//		'DECLARE @ID_INSERTED TABLE (Id INT) INSERT INTO ProductionMachineParameters (IdLineStation, MachineNumber, IdComposedPart, ParamsData, CRC_Sum) OUTPUT INSERTED.ID INTO @ID_INSERTED VALUES ({IdLineStation}, {MachineNumber}, {IdComposedPart}, ( CONVERT ( VARBINARY({iStructDataSize}), {astStructRawData}) ), {iCRC16sum}) SELECT Id FROM @ID_INSERTED';
//		'DECLARE @ID_INSERTED TABLE (Id INT) INSERT INTO ProductionMachineParameters (IdLineStation, MachineNumber, IdComposedPart, ParamsData, CRC_Sum) OUTPUT INSERTED.ID INTO @ID_INSERTED VALUES ({IdLineStation}, {MachineNumber}, (SELECT IdOutComposedPart FROM ProductionLineStation WHERE Id ={IdLineStation}), {astStructRawData}, {iCRC16sum}) SELECT Id FROM @ID_INSERTED';
//		'DECLARE @ID_INSERTED TABLE (Id INT) INSERT INTO ProductionMachineParameters (IdLineStation, MachineNumber, IdComposedPart, ParamsData, CRC_Sum) OUTPUT INSERTED.ID INTO @ID_INSERTED VALUES ({IdLineStation}, {MachineNumber}, (SELECT IdOutComposedPart FROM ProductionLineStation WHERE Id ={IdLineStation}), CAST({astStructRawData} AS VARBINARY({iStructDataSize})), {iCRC16sum}) SELECT Id FROM @ID_INSERTED';
//		'DECLARE @ID_INSERTED TABLE (Id INT) INSERT INTO ProductionMachineParameters (IdLineStation, MachineNumber, IdComposedPart, ParamsData, CRC_Sum) OUTPUT INSERTED.ID INTO @ID_INSERTED VALUES ({IdLineStation}, {MachineNumber}, {IdComposedPart}, {astStructRawData}, {iCRC16sum}) SELECT Id FROM @ID_INSERTED';
//		'DECLARE @ID_INSERTED TABLE (Id INT) INSERT INTO ProductionMachineParameters (IdLineStation, MachineNumber, IdComposedPart, ParamsData, CRC_Sum) OUTPUT INSERTED.ID INTO @ID_INSERTED VALUES ({IdLineStation}, {MachineNumber}, {IdComposedPart}, CAST({astStructRawData} AS VARBINARY({iStructDataSize})), {iCRC16sum}) SELECT Id FROM @ID_INSERTED';
//		'UPDATE [dbo].[ProductionMachineParameters] SET Active = 0 WHERE IdLineStation = {IdLineStation} AND IdComposedPart = {IdComposedPart} DECLARE @ID_INSERTED TABLE (Id INT) INSERT INTO [dbo].[ProductionMachineParameters] (IdLineStation, MachineNumber, IdComposedPart,ParamsData,CRC_Sum,ParamsSizeInBytes) OUTPUT INSERTED.ID INTO @ID_INSERTED VALUES ({IdLineStation}, {MachineNumber}, {IdComposedPart}), CAST( {astStructRawData} AS VARBINARY(';
	
		stSqlComandData.pReturnedData := ADR(diMachineParamsInsertId);
		stSqlComandData.uiReturnedDataSize := SIZEOF(diMachineParamsInsertId);
		stSqlComandData.bSQL_OK := stSqlComandData.bSQL_Done := FALSE;
		// Próba dodania komendy do kolejki
		IF I_SqlCore <> 0 AND_THEN I_SqlCore.mAddCmdToQueue(ADR(stSqlComandData)) THEN
			bCmdSended := bReturnDataBusy := bReturnDataReserved_InsMachParams := TRUE;		// Zajęcie struktury danych
			diMachineParamsInsertId := 0;
		ELSE
			bResultOk := FALSE;
			nErrorID:=nPIM_ErrorCodes.ParamsSaveToDB_Error;
			m_SqlInsMachineParamsData := bCmdAddError := TRUE;
		END_IF
	ELSIF stSqlComandData.bSQL_Done THEN
		IF stSqlComandData.bSQL_OK THEN
			diParamsId := diMachineParamsInsertId;
		ELSE
			nErrorID:=nPIM_ErrorCodes.ParamsSaveToDB_Error;
		END_IF
		bInsMachineParamsData := TRUE;	// Odśwież parametrów w strukturze PIM, skasowanie zmiennej bCmdSended
		bResultOK := stSqlComandData.bSQL_OK;
		m_SqlInsMachineParamsData := bUpdateData := TRUE;
	END_IF
END_IF
bProcessing := bCmdSended AND NOT stSqlComandData.bSQL_Done;
END_METHOD

// Zapis do DB statusu ostatniej operacji - gdy rozkaz zostanie wykonany zwraca TRUE
METHOD m_SqlSelInsStatus : BOOL
VAR_INPUT
	bStatus:BOOL:= FALSE;		// Status operacji do zapisania
	sErrCode:STRING(10);		// kod błędu - tylko jeśli status  FALSE
	bSustein:BOOL:= FALSE;		// Jeśli TRUE po wywołaniu przez FbMaszyny wykonwyanie rozkazu przerzucone na fbStation (wysyłanie rozkazu w tle)- ustawiana odpowiednia flaga 
END_VAR
VAR_OUTPUT
	bProcessing:BOOL;			// Przetwarzanie rozkazu trwa (rozkaz dodany do kolejki)
	bResultOK:BOOL;				// Wynik wykonania rozkazu (do sprawdzenia gdy metoda zwróci TRUE)
	liStatusId:LINT;			// Id statusu części w DB
END_VAR

VAR
	byStatus: BYTE;
	byIsHidden: BYTE;
END_VAR
// Rezerwacja struktury danych dla zapytania
IF NOT bReturnDataBusy OR bReturnDataReserved_InsOperStat AND stRetDataLineStation.IdStacji <> 0 THEN
	IF NOT bCmdSended THEN	// Przygotowanie danych do zapytania
		stSqlComandData.nCmdState:= nSQL_CmdExecState.New;
		stSqlComandData.nCmdType:=nSQL_CmdTypes.SelInsStatusOfOperation;
		stSqlComandData.byExecutingNodeNb:=0;
		stSqlComandData.bWaitForDataReturn:=TRUE;
	
		stSqlComandData.stStatusSaveParams.didLineStation := stRetDataLineStation.IdStacji;
		stSqlComandData.stStatusSaveParams.byStatus := BOOL_TO_BYTE(bStatus);
		IF bStatus THEN
			stSqlComandData.stStatusSaveParams.byIsHidden := BOOL_TO_BYTE(bIsHidden);
		ELSE
			stSqlComandData.stStatusSaveParams.byIsHidden := 0;
		END_IF
		stSqlComandData.stStatusSaveParams.byIsTestMode := BOOL_TO_BYTE(stPimInOut.bTestMode);
		stSqlComandData.stStatusSaveParams.iMachineNb := iMachineNumber;
		stSqlComandData.stStatusSaveParams.lrQuantity := 1.0;
		byStatus := BOOL_TO_BYTE(bStatus);
		byIsHidden := BOOL_TO_BYTE(bIsHidden);
(*		IF bStatus THEN
			sFormat := 'DECLARE @ID_TABLE TABLE (Id bigint) insert into [dbo].[ProductionMachinePartsStatuses] (IdLineStation, Status, MachineNumber, IsHidden) output inserted.id into @ID_TABLE values (%d, %d, %d, %d) SELECT Top(1) Id FROM @ID_TABLE';
				fbFormatStr2(pFormatString := ADR(sFormat),
				arg1:= F_DINT(stRetDataLineStation.IdStacji),
				arg2:= F_BYTE(byStatus),
				arg3:= F_INT(iMachineNumber),
				arg4:= F_BYTE(byIsHidden),
				pDstString := ADR(stSqlComandData.sCmdExpression), nDstSize := SIZEOF(stSqlComandData.sCmdExpression));
		ELSE
			sFormat := 'DECLARE @ID_TABLE TABLE (Id bigint) insert into [dbo].[ProductionMachinePartsStatuses] (IdLineStation, Status, MachineNumber, IsHidden) output inserted.id into @ID_TABLE values (%d, %d, %d, %d) DECLARE @statusId bigint = (SELECT Top(1) Id FROM @ID_TABLE) INSERT INTO [dbo].[ProductionMachinePartsStatusDefectRelation] (IdPartStatus, IdMachineError) values (@statusId, (SELECT Id FROM [dbo].[ProductionMachineError] WHERE Active = 1 AND Code = $'%s$')) SELECT @statusId';
				fbFormatStr2(pFormatString := ADR(sFormat),
				arg1:= F_DINT(stRetDataLineStation.IdStacji),
				arg2:= F_BYTE(byStatus),
				arg3:= F_INT(iMachineNumber),
				arg4:= F_BYTE(byIsHidden),
				arg5:= F_STRINGEx(sErrCode),
				pDstString := ADR(stSqlComandData.sCmdExpression), nDstSize := SIZEOF(stSqlComandData.sCmdExpression));
		END_IF
*)		
		bLastStatus := bStatus;
		sLastErrCode:= sErrCode;
		stSqlComandData.pReturnedData := ADR(liLPartStatusId);
		stSqlComandData.uiReturnedDataSize := SIZEOF(liLPartStatusId);
		bStatusSavedOK := stSqlComandData.bSQL_OK := stSqlComandData.bSQL_Done := FALSE;
		// Próba dodania komendy do kolejki
		IF I_SqlCore <> 0 AND_THEN I_SqlCore.mAddCmdToQueue(ADR(stSqlComandData)) THEN
			bCmdSended := bReturnDataBusy := bReturnDataReserved_InsOperStat := TRUE;		// Zajęcie struktury danych
			liLPartStatusId := 0;
			bInsertStatus S= bSustein;
		ELSE
			bResultOk := FALSE;
			m_SqlSelInsStatus := bCmdAddError := TRUE;
		END_IF
	ELSIF stSqlComandData.bSQL_Done THEN
		IF stSqlComandData.bSQL_OK THEN
			liStatusId := liLPartStatusId;	// Uaktualnij zmienną wyjściową
		END_IF
		bInsertStatus := TRUE;	// Odśwież parametrów w strukturze PIM, skasowanie zmiennej bCmdSended
		bResultOK := stSqlComandData.bSQL_OK;
		m_SqlSelInsStatus := bUpdateData := TRUE;
	END_IF
END_IF
bProcessing := bCmdSended AND NOT stSqlComandData.bSQL_Done;
END_METHOD

// Pobranie z DB statusu ostatniej operacji dla danego DM z poprzedniego stanowiska - gdy rozkaz zostanie wykonany zwraca TRUE
METHOD m_SqlSelLastOperationStatus : BOOL
VAR_INPUT
	sCodeDM:STRING(255);		// Identyfikator części (kod DataMatrix)
END_VAR
VAR_OUTPUT
	bProcessing:BOOL;			// Przetwarzanie rozkazu trwa (rozkaz dodany do kolejki)
	bResultOK:BOOL;				// Wynik wykonania rozkazu (do sprawdzenia gdy metoda zwróci TRUE)
	bPrevOperStat:BOOL;			// Status ostatniej operacji na poprzednim stanowisku
END_VAR
// Rezerwacja struktury danych dla zapytania
IF NOT bReturnDataBusy OR bReturnDataReserved_SelLastOperStat THEN
	IF NOT bCmdSended THEN
		// Przygotowanie danych do zapytania
		stSqlComandData.nCmdState:= nSQL_CmdExecState.New;
		stSqlComandData.nCmdType:=nSQL_CmdTypes.SelLastOperationStatus;
		stSqlComandData.byExecutingNodeNb:=0;
		stSqlComandData.bWaitForDataReturn:=TRUE;

		sFormat := 'SELECT TOP(1) PMPS.Status FROM [dbo].[ProductionMachinePartsStatuses] PMPS INNER JOIN [dbo].[ProductionLineStation] PLS ON PLS.Id = PMPS.IdLineStation WHERE PLS.Active = 1 AND PMPS.NumberId = $'%s$' AND PLS.Name = $'%s$' AND PMPS.IsHidden = 0 ORDER BY PMPS.Date desc';
		fbFormatStr2(pFormatString := ADR(sFormat),
			arg1:= F_STRINGEx(sCodeDM),
			arg2:= F_STRINGEx(sPrevStationName),
			pDstString := ADR(stSqlComandData.sCmdExpression), nDstSize := SIZEOF(stSqlComandData.sCmdExpression));
			
		sLastDMCode := sCodeDM;
		stSqlComandData.pReturnedData := ADR(bPreviousOperationStatus);
		stSqlComandData.uiReturnedDataSize := SIZEOF(bPreviousOperationStatus);
		stSqlComandData.bSQL_OK := stSqlComandData.bSQL_Done := FALSE;
		// Próba dodania komendy do kolejki
		IF I_SqlCore <> 0 AND_THEN I_SqlCore.mAddCmdToQueue(ADR(stSqlComandData)) THEN
			bCmdSended := 	bReturnDataBusy := bReturnDataReserved_SelLastOperStat := TRUE;		// Zajęcie struktury danych
			bPreviousOperationStatus := FALSE;
		ELSE
			bResultOk := FALSE;
			m_SqlSelLastOperationStatus := bCmdAddError := TRUE;
		END_IF
	ELSIF stSqlComandData.bSQL_Done THEN		// Komenda została wykonana, sprawdzenie rezultatu
		IF stSqlComandData.bSQL_OK THEN
			bPrevOperStat := bPreviousOperationStatus;	// Uaktualnij zmienną wyjściową
		END_IF
		bSelPreviousStatus := TRUE;	// Odśwież parametrów w strukturze PIM, skasowanie zmiennej bCmdSended
		bResultOK := stSqlComandData.bSQL_OK;
		m_SqlSelLastOperationStatus := bUpdateData := TRUE;
	END_IF
END_IF
bProcessing := bCmdSended AND NOT stSqlComandData.bSQL_Done;
END_METHOD

// Pobranie z DB ID stanowiska - gdy rozkaz zostanie wykonany zwraca TRUE
METHOD PRIVATE m_SqlSelLineStationId : BOOL
VAR_INPUT
END_VAR
VAR_OUTPUT
	bProcessing:BOOL;			// Przetwarzanie rozkazu trwa (rozkaz dodany do kolejki)
	bResultOK:BOOL;				// Wynik wykonania rozkazu (do sprawdzenia gdy metoda zwróci TRUE)
	diStationId:DINT;			// Identyfikator stanowiska
	liIdCompossedPart:LINT;		// Identyfikator części wyjściowej
	bAutoSaveErrors:BOOL;		// Auto zapis błędów
	bAutoControlMachineParams:BOOL;		// Kontrola parametrów maszyny
	wCrcSumInDB:WORD;			// Suma CRC aktualnych parametrów maszyny dla złożenia wyjściowego
END_VAR
// Rezerwacja struktury danych dla zapytania
IF NOT bReturnDataBusy OR bReturnDataReserved_StationId THEN
	IF NOT bCmdSended THEN
		// Przygotowanie danych do zapytania
		stSqlComandData.nCmdState:= nSQL_CmdExecState.New;
		stSqlComandData.nCmdType:=nSQL_CmdTypes.SelStationId;
		stSqlComandData.byExecutingNodeNb:=0;
		stSqlComandData.bWaitForDataReturn:=TRUE;
		sFormat := 'SELECT PL.Id, PLS.Id, PLS.IsAutoSaveErrors, PLS.IsEol, PLS.IdOutComposedPart, PMP.CRC_Sum, PCP.CodeNumber FROM [dbo].[ProductionLineStation] PLS INNER JOIN [dbo].[ProductionLine] PL on PLS.IdLine=PL.Id LEFT JOIN [dbo].[ProductionMachineParameters] PMP on PLS.Id=PMP.IdLineStation AND PLS.IdOutComposedPart=PMP.IdComposedPart AND PMP.MachineNumber=%d AND PMP.Active=1 LEFT JOIN [dbo].[ProductionComposedPart] PCP on PLS.IdOutComposedPart=PCP.Id AND PCP.Active=1 WHERE PL.Active = 1 AND PL.Name = $'%s$' AND PLS.Name = $'%s$' AND PLS.Active=1';
		fbFormatStr2(pFormatString := ADR(sFormat),
			arg1:= F_INT(iMachineNumber),
			arg2:= F_STRINGEx(sLineName),
			arg3:= F_STRINGEx(sStationName),
			pDstString := ADR(stSqlComandData.sCmdExpression), nDstSize := SIZEOF(stSqlComandData.sCmdExpression));
		stSqlComandData.pReturnedData := ADR(stRetDataLineStation);
		stSqlComandData.uiReturnedDataSize := SIZEOF(stRetDataLineStation);
		stSqlComandData.bSQL_OK := stSqlComandData.bSQL_Done := FALSE;
		// Próba dodania komendy do kolejki
		IF I_SqlCore <> 0 AND_THEN I_SqlCore.mAddCmdToQueue(ADR(stSqlComandData)) THEN
			bSelectStationId := bCmdSended := bReturnDataBusy := bReturnDataReserved_StationId := TRUE;		// Zajęcie struktury danych
			diStationId := 0;
			MEMSET(destAddr := ADR(stRetDataLineStation), n := SIZEOF(stRetDataLineStation), fillByte:= 0);		// Czyszczenie danych 
		ELSE
			bResultOk := FALSE;
			m_SqlSelLineStationId := bCmdAddError := TRUE;
		END_IF
	ELSIF stSqlComandData.bSQL_Done THEN
		IF stSqlComandData.bSQL_OK THEN
			diStationId := stRetDataLineStation.IdStacji;	// Uaktualnij zmienne wyjściowe
			liIdCompossedPart := stRetDataLineStation.IdOutComposedPart;
			bAutoSaveErrors := stRetDataLineStation.AutoSaveErrors;
			bAutoControlMachineParams := FALSE;// stRetDataLineStation.AutoControlMachineParams; 
			wCrcSumInDB:= stRetDataLineStation.CrcSumOfParams;
		END_IF
		bSelectStationId := bUpdateData := TRUE;	// Odświeżenie parametrów w strukturze PIM w cżęści głównej bloku funkcyjnego, skasowanie zmiennej bCmdSended
		bResultOK := stSqlComandData.bSQL_OK;
		m_SqlSelLineStationId := TRUE;
	END_IF
END_IF
bProcessing := bCmdSended AND NOT stSqlComandData.bSQL_Done;
END_METHOD

// Pobranie z DB sumy CRC parametrów pracy maszyny - gdy rozkaz zostanie wykonany zwraca TRUE
METHOD PRIVATE m_SqlSelMachineParamsCRC : BOOL
VAR_INPUT
	liIdCompossedPart:LINT;		// Identyfikator części wyjściowej dla którego powinna zostać pobrana suma 
END_VAR
VAR_OUTPUT
	bProcessing:BOOL;		// Przetwarzanie rozkazu trwa (rozkaz dodany do kolejki)
	bResultOK:BOOL;			// Wynik wykonania rozkazu (do sprawdzenia gdy metoda zwróci TRUE)
	diStationId:DINT;		// Identyfikator stanowiska
	wCrcFromDb:WORD;		// Suma CRC pobrana z DB
END_VAR
// Sprawdzenie danych wejściowych - jeśli błędne przerwij procedure
IF liIdCompossedPart = 0 OR stRetDataLineStation.IdStacji = 0 THEN
	m_SqlSelMachineParamsCRC := TRUE;
	bResultOK := FALSE;
	RETURN;
END_IF

// Rezerwacja struktury danych dla zapytania
IF NOT bReturnDataBusy OR bReturnDataReserved_SelMachParamsCRC THEN
	IF NOT bCmdSended THEN
		// Przygotowanie danych do zapytania
		stSqlComandData.nCmdState:= nSQL_CmdExecState.New;
		stSqlComandData.nCmdType:=nSQL_CmdTypes.SelMachineParamsCRC;
		stSqlComandData.byExecutingNodeNb:=0;
		stSqlComandData.bWaitForDataReturn:=TRUE;
	
		
		sFormat := 'SELECT CRC_Sum, FROM [dbo].[ProductionMachineParameters] WHERE Active = 1 AND IdLineStation = %d AND MachineNumber = %d AND IdComposedPart = %d';
		fbFormatStr2(pFormatString := ADR(sFormat),
			arg1:= F_DINT(stRetDataLineStation.IdStacji),
			arg2:= F_INT(iMachineNumber),
			arg3:= F_LINT(stRetDataLineStation.IdOutComposedPart),
			pDstString := ADR(stSqlComandData.sCmdExpression), nDstSize := SIZEOF(stSqlComandData.sCmdExpression));

(*		stSqlComandData.sCmdExpression := 'SELECT CRC_Sum, FROM [dbo].[ProductionMachineParameters] WHERE Active = 1 AND IdLineStation = {IdLineStation} AND MachineNumber = {MachineNumber} AND IdComposedPart = {IdComposedPart}';
		stSqlComandData.stCmdData.IdLineStation := stRetDataLineStation.IdStacji;
		stSqlComandData.stCmdData.MachineNumber := iMachineNumber;
		IF liIdCompossedPart = 0 THEN			// Jeśli 0 pobiera dla aktualnie produkowanego, można też pobrać dla konkretnego Id
			stSqlComandData.stCmdData.IdComposedPart := stRetDataLineStation.IdOutComposedPart;
		ELSE
			stSqlComandData.stCmdData.IdComposedPart := liIdCompossedPart;
		END_IF	*)
		stSqlComandData.pReturnedData := ADR(wCrcSumInDb);
		stSqlComandData.uiReturnedDataSize := SIZEOF(wCrcSumInDb);
		stSqlComandData.bSQL_OK := stSqlComandData.bSQL_Done := FALSE;
		// Próba dodania komendy do kolejki
		IF I_SqlCore <> 0 AND_THEN I_SqlCore.mAddCmdToQueue(ADR(stSqlComandData)) THEN
			bCmdSended := bReturnDataBusy := bReturnDataReserved_SelMachParamsCRC := TRUE;		// Zajęcie struktury danych
			wCrcSumInDb := 0;
		ELSE
			bResultOk := FALSE;
			m_SqlSelMachineParamsCRC := bCmdAddError := TRUE;
		END_IF
	ELSIF stSqlComandData.bSQL_Done THEN
		IF stSqlComandData.bSQL_OK THEN
			wCrcFromDb := wCrcSumInDb;	// Uaktualnij zmienne wyjściowe
		END_IF
		m_SqlSelMachineParamsCRC := TRUE;	// Odświeżenie parametrów w strukturze PIM w cżęści głównej bloku funkcyjnego, skasowanie zmiennej bCmdSended
		bResultOK := stSqlComandData.bSQL_OK;
		m_SqlSelMachineParamsCRC := bUpdateData := TRUE;
	END_IF
END_IF
bProcessing := bCmdSended AND NOT stSqlComandData.bSQL_Done;
END_METHOD

// Pobranie z DB parametrów pracy maszyny - gdy rozkaz zostanie wykonany zwraca TRUE
METHOD m_SqlSelMachineParamsData : BOOL
VAR_INPUT
	diParamsId:DINT:=0;				// Jeśli 0 - pobiera parametry dla aktualnego złożenia, jeśli <>0 wtedy pobiera zestaw parametrów o danym Id
	pParamsData:POINTER TO BYTE;	// Wskaźnik do struktury parametrów maszyny
	uiParamsDataSize:UINT;			// Rozmiar struktury danych parametrów maszyny
END_VAR
VAR_OUTPUT
	bProcessing:BOOL;				// Przetwarzanie rozkazu trwa (rozkaz dodany do kolejki)
	bResultOK:BOOL;					// Wynik wykonania rozkazu (do sprawdzenia gdy metoda zwróci TRUE)
	bNoMatchingParams:BOOL;			// Błąd - brak pasujących parametrów w DB
	bParametersUpdated:BOOL;		// Parametry maszyny uaktualnione
//	pParamsData: POINTER TO BYTE;
END_VAR
(*
Zapis i odczyt parametrów kontroluje blok klienta PIM, struktura w bloku przechowywana jest jako wskaźnik więc nie jest konieczne powiązanie ze strukturą parametrów maszyny.
Metoda pobiera z DB najnowszy zestaw parametrów lub zestaw o danym Id (jeśli Id nie jest równe 0), sprawdza czy rozmiary oraz suma CRC są zgodne - jeśli są przepisuje pobrane dane do wskaźnika wejściowego.
Jeśli nie co zrobić - może pytanie do użytkownika (przez komendy PIM) "Rozmiar/wartość danych niezgodna - pomiń lub nadpisz" - użytkownik wybierze odpowiendią opcje która zostanie zwrócona do PLC.
Póki co następuje automatyczne przepisanie niekompletnych lub niezgodnych parametrów.
*)

// Sprawdzenie danych wejściowych - jeśli błędne przerwij procedure
IF pParamsData = 0 OR uiParamsDataSize = 0 OR SEL(diParamsId=0, stRetDataLineStation.IdStacji = 0, stRetDataLineStation.IdStacji = 0 OR stRetDataLineStation.IdOutComposedPart = 0) THEN
	m_SqlSelMachineParamsData := TRUE;
	bResultOK := FALSE;
	RETURN;
END_IF

// Rezerwacja struktury danych dla zapytania
IF NOT bReturnDataBusy OR bReturnDataReserved_SelMachParams THEN
	IF NOT bCmdSended THEN	// Przygotowanie danych do zapytania
		stSqlComandData.nCmdState:= nSQL_CmdExecState.New;
		stSqlComandData.nCmdType:=nSQL_CmdTypes.SelMachineParams;
		stSqlComandData.byExecutingNodeNb:=0;
		
	(*	stSqlComandData.bWaitForDataReturn:=TRUE;
		IF diParamsId <> 0 THEN		// Rodzaj zapytania zależy od tego po czym chcemy wyszukiwać zestawy parametrów 
			stSqlComandData.sCmdExpression :=  'SELECT ParamsData, CRC_Sum, ParamsSizeInBytes FROM [dbo].[ProductionMachineParameters] WHERE Id = {IdLineStation}';
			stSqlComandData.stCmdData.IdLineStation := diParamsId;
		ELSE
			stSqlComandData.sCmdExpression :=  'SELECT ParamsData, CRC_Sum, ParamsSizeInBytes FROM [dbo].[ProductionMachineParameters] WHERE Active = 1 AND MachineNumber = {MachineNumber} AND IdLineStation = {IdLineStation} AND IdComposedPart = {IdComposedPart}';
			stSqlComandData.stCmdData.MachineNumber := iMachineNumber;
			stSqlComandData.stCmdData.IdLineStation := stRetDataLineStation.IdStacji;
			stSqlComandData.stCmdData.IdComposedPart := stRetDataLineStation.IdOutComposedPart;
		END_IF	*)
		stSqlComandData.pReturnedData := ADR(stRetDataMachParams);
		stSqlComandData.uiReturnedDataSize := SIZEOF(stRetDataMachParams);
		stSqlComandData.bSQL_OK := stSqlComandData.bSQL_Done := FALSE;
		// Próba dodania komendy do kolejki
		IF I_SqlCore <> 0 AND_THEN  I_SqlCore.mAddCmdToQueue(ADR(stSqlComandData)) THEN
			bCmdSended := bReturnDataBusy := bReturnDataReserved_SelMachParams := TRUE;		// Zajęcie struktury danych
			MEMSET(destAddr := ADR(stRetDataMachParams), n := SIZEOF(stRetDataMachParams), fillByte:= 0);		// Czyszczenie danych 
		ELSE
			bResultOk := FALSE;
			m_SqlSelMachineParamsData := bCmdAddError := TRUE;
		END_IF
	ELSIF stSqlComandData.bSQL_Done THEN	// Przetwarzanie zapytania SQL zakończone 
		IF stSqlComandData.bSQL_OK THEN
			IF stRetDataMachParams.DataSize = UINT_TO_INT(uiParamsDataSize) THEN	// Rozmiar parametrów zgodny
				IF INT_TO_WORD(stRetDataMachParams.CRC16sum) = F_DATA_TO_CRC16_CCITT(pData := ADR(stRetDataMachParams.StructRawData), cbData := INT_TO_UDINT(stRetDataMachParams.DataSize), crc:= 0) THEN
					MEMCPY(srcAddr := ADR(stRetDataMachParams.StructRawData), destAddr := pParamsData, n:= uiParamsDataSize);
					bParametersUpdated := TRUE;
				ELSE		// Niezgodne sumy CRC - raczej niemożliwe
					mNewlnternalEvent(nInputErrorID := nPIM_ErrorCodes.ParamsMismatchPLCandDB, nEventType := nPIM_EventClasses.Alarm, tMessageTime := T#0S);
					MEMCPY(srcAddr := ADR(stRetDataMachParams.StructRawData), destAddr := pParamsData, n:= uiParamsDataSize);
				END_IF
			ELSE
				mNewlnternalEvent(nInputErrorID := nPIM_ErrorCodes.ParamsMismatchPLCandDB, nEventType := nPIM_EventClasses.Alarm, tMessageTime := T#0S);
				MEMSET(destAddr := pParamsData, n := uiParamsDataSize, fillByte:= 0);		// Czyszczenie danych parametrów
				MEMCPY(srcAddr := ADR(stRetDataMachParams.StructRawData), destAddr := pParamsData, n:= MIN(uiParamsDataSize,INT_TO_UINT(stRetDataMachParams.DataSize)));
			END_IF
		ELSE	// Jeśli nie zwrócono żadnego rekordu brak pasujących parametrów - trzeba najpierw przesłać parametry do DB
			mNewlnternalEvent(nInputErrorID := nPIM_ErrorCodes.NoMatchingParamsForComponent, nEventType := nPIM_EventClasses.Alarm, tMessageTime := T#0S);
			bNoMatchingParams := TRUE;	;
		END_IF
		bSelMachineParamsData := TRUE;	// Odświeżenie parametrów w strukturze PIM, skasowanie zmiennej bCmdSended
		bResultOK := stSqlComandData.bSQL_OK;
		m_SqlSelMachineParamsData := bUpdateData := TRUE;
	END_IF
END_IF
pParamsData := ADR(stRetDataMachParams.StructRawData);
bProcessing := bCmdSended AND NOT stSqlComandData.bSQL_Done;
END_METHOD

ACTION ACT_PimCmdsHandling:
// TImer gotowości PIMu (komunikacja itp jest OK)
fbTOF_PimWorking(IN:= FALSE, PT:= T#5M, Q=> bPIM_Working);		// TImer o gotowości systemu PIM

//Obsługa komunikatów z PIMu
IF stPimInOut.sCmdPIM2PLC <> '' AND NOT bCmdReaded THEN
	fbLogger.mAddLine(sTextToSave := CONCAT(STR1:= 'CmdRecived- ', STR2:=stPimInOut.sCmdPIM2PLC));
	sCmdToSendToMachine := sStringToParse := F_ToLCase(stPimInOut.sCmdPIM2PLC);
	WHILE sStringToParse <> '' DO
		sActCmd := fPIM_GetCmdPar(sParseString := sStringToParse);
		IF sActCmd = 'lifebit' THEN
			fbTOF_PimWorking(IN:= TRUE);
		ELSIF sActCmd = 'sendmachineparamstodb' THEN			// Zapisuje w bazie danych parametry pracy dla aktualnego złożenia jako aktywne 
			bMachParamsSendToDB:= TRUE;
		ELSIF sActCmd = 'readmachineparamsfromdb' THEN
			bMachParamsReadFromDB := TRUE;	// Wymuszenie pobrania parametrów z bazy danych
			bMachineParamsOK := FALSE;		// Zatrzymanie pracy na czas pobrania elementów
		ELSIF sActCmd = 'retool' THEN		// Pobiera z bazy danych parametry dla danego złożenia
			sActCmd := fPIM_GetCmdPar(sParseString := sStringToParse);
			liRetoolParamsIdFromPIM:= STRING_TO_LINT(sActCmd);
//			bRetool := TRUE;	// Wymuszenie pobrania parametrów z bazy danych
//			bMachineParamsOK := FALSE;		// Zatrzymanie pracy na czas pobrania elementów
		ELSIF sActCmd = 'newboxout' THEN
			iOutBoxQty:= STRING_TO_INT(fPIM_GetCmdPar(sParseString := sStringToParse));
			iOutBoxTargetQty:= STRING_TO_INT(fPIM_GetCmdPar(sParseString := sStringToParse));
		ELSIF sActCmd = 'nokreported' THEN	// Zgłoszenie po wykonaniu operacji - do ustalenia źródło zgłoszenia
			sActCmd := fPIM_GetCmdPar(sParseString := sStringToParse);				
			IF sActCmd = 'fprevstation' THEN
				nReoprtedNokSource:= nPIM_ReportedNokSource.FromPrevStation;
			ELSIF sActCmd = 'fmach' THEN
				nReoprtedNokSource:= nPIM_ReportedNokSource.FromMach;				
			ELSIF sActCmd = 'fbox' THEN
				nReoprtedNokSource:= nPIM_ReportedNokSource.FromBox;
			ELSE
				nReoprtedNokSource:= nPIM_ReportedNokSource.Error_UnknownSource;			
			END_IF
		ELSIF sActCmd = 'rework' THEN
			IF fPIM_GetCmdPar(sParseString := sStringToParse) = 'true' THEN
				nReworkMenuStatus := nPIM_ReworkSelect.yes;
				iCtr_PIM_ReworkYes := iCtr_PIM_ReworkYes + 1;
				iCtr_PIM_PartsNOK := LIMIT(0,iCtr_PIM_PartsNOK - 1,32767);
			ELSE
				nReworkMenuStatus := nPIM_ReworkSelect.no;
			END_IF
		ELSIF sActCmd = 'logged' THEN
			sUserRole:= fPIM_GetCmdPar(sParseString := sStringToParse);
			sUserLang:= fPIM_GetCmdPar(sParseString := sStringToParse);
		ELSIF sActCmd = '' THEN
			MEMMOVE(srcAddr := ADR(asUnsuportedCmds[1]), destAddr := ADR(asUnsuportedCmds[2]), n := 4*SIZEOF(asUnsuportedCmds[1]));
			asUnsuportedCmds[1] := 'EmptyString';
		ELSE
			MEMMOVE(srcAddr := ADR(asUnsuportedCmds[1]), destAddr := ADR(asUnsuportedCmds[2]), n := 4*SIZEOF(asUnsuportedCmds[1]));
			asUnsuportedCmds[1] := sActCmd;
		END_IF
	END_WHILE
	bCmdReaded := TRUE;
ELSE
	stPimInOut.sCmdPIM2PLC := '';
	ACT_UpdatePimOutput();
	bCmdReaded := FALSE;
	nReoprtedNokSource:= nPIM_ReportedNokSource.none;
	nReworkMenuStatus := nPIM_ReworkSelect.none;
END_IF

//Obsługa komunikatów z PIMu
fbTON_CmdPLC2PIM_Reset(IN:= stPimInOut.sCmdPLC2PIM <> '', PT:= T#100MS);
IF fbTON_CmdPLC2PIM_Reset.Q THEN
	stPimInOut.sCmdPLC2PIM := '';
	bCmdPlc2PimSended := FALSE;
END_IF
bCmdPlc2PimSended R= stPimInOut.sCmdPLC2PIM = '';

(*	Komendy do wysłania:
	- Wyloguj użytkownika?
	- Zgłoś usterkę maszyny
*)
END_ACTION

ACTION ACT_SqlDataReturnCmd:

{warning 'Uzupełnić działanie LifeBita, Timeoutu'}
fbTON_CmdHangedUp(IN:= bReturnDataBusy AND NOT stSqlComandData.bSQL_Done AND I_SqlCore.IsCoreWork(), PT:= T#20S);
IF fbTON_CmdHangedUp.Q THEN
	fbTON_CmdHangedUp(IN:= FALSE);
	stSqlComandData.bSQL_Done := TRUE;
	stSqlComandData.bSQL_Busy := stSqlComandData.bSQL_OK := FALSE;
	fbLogger.mAppendCurrentLine(bBreakLine := TRUE, sAddSep := '', sAppendText:= CONCAT('Sql command Hungedup, service reset- Cmd State ',INT_TO_STRING(stSqlComandData.nCmdState)));
	uiCtr_CmdReset:= uiCtr_CmdReset +1; 
END_IF

stSqlComandData.bSQL_LifeBit := FALSE;

IF bTestAdditionalErrorSave THEN
	bTestAdditionalErrorSave := bTestResult:= FALSE;
	bTestResult:= m_SqlInsAdditionalError(sErrCode := sLastErrCode);
ELSIF bTestComprAirCtrSave THEN
	bTestComprAirCtrSave := bTestResult:= FALSE;
	bTestResult:= m_SqlInsCompressedAirConsumption(rActCompressedAirConsumption := 9.99);
ELSIF bTestEnergyCtrSave THEN
	bTestEnergyCtrSave := bTestResult:= FALSE;
	bTestResult:= m_SqlInsEnergyConsumption(rActEnergyConsumption := 9.99);
ELSIF bTestDefectRealtionSave THEN
	bTestDefectRealtionSave:= bTestResult := FALSE;
	bTestResult:= m_SqlInsDefectRelation(sErrCode := '54');	
END_IF

// Jeśli chcemy serwisowo sprawdzić działanie funkcji ustawić zmienne wejściowe w odpowiedni sposób oraz ustawić zmienną w If np. bSelectStationId
IF bSelectStationId THEN
	IF NOT bUpdateData THEN
		m_SqlSelLineStationId(bProcessing => bPimCmdProcessing);
	END_IF
	IF stSqlComandData.bSQL_Done THEN
		IF stSqlComandData.bSQL_OK THEN		// Pobranie danych OK
		//	stRetDataLineStation.AutoControlMachineParams := FALSE;
			fbLogger.mAddLine(sTextToSave := CONCAT(STR1:= 'RecvStationId- ', STR2:= DINT_TO_STRING(stRetDataLineStation.IdStacji)));
			stStationStatus.stStationSqlData := stRetDataLineStation; 
		ELSE 
			fbLogger.mAddLine(sTextToSave := 'RecvStationId rvc error');
		END_IF
		bPimCmdProcessing := bCmdSended := bSelectStationId := FALSE;
		bReturnDataBusy := bReturnDataReserved_StationId := FALSE;
	//	MEMSET(destAddr := ADR(stDBCmdData), n := SIZEOF(stDBCmdData), fillByte:= 0);		// Czyszczenie danych zapytania
	ELSIF NOT bPimCmdProcessing THEN
		bCmdSended := bSelectStationId := FALSE;
		bReturnDataBusy := bReturnDataReserved_StationId := FALSE;		
	END_IF
END_IF

IF bInsertStatus THEN 
	IF NOT bUpdateData THEN
		m_SqlSelInsStatus(bStatus:=bLastStatus , sErrCode:= sLastErrCode, bSustein := FALSE, bProcessing => bPimCmdProcessing);
	END_IF
	IF stSqlComandData.bSQL_Done THEN	
		IF stSqlComandData.bSQL_OK THEN
			bStatusSavedOK := TRUE;
		
			iCtr_StatusSaveOK := iCtr_StatusSaveOK + 1; 
			mSendCmdToPIM(sCmd := CONCAT(STR1:='StatusId:', STR2:= LINT_TO_STRING(liLPartStatusId)));
			IF bLastStatus THEN
		
				fbLogger.mAddLine(sTextToSave := CONCAT(STR1:= 'Status OK saved, StatusId- ', STR2:= LINT_TO_STRING(liLPartStatusId)));
				iCtr_PIM_PartsOK := iCtr_PIM_PartsOK +1;
			ELSE
				stPimInOut.sStatusNokAndErrorID := CONCAT(STR1:= LINT_TO_STRING(liLPartStatusId), STR2:= CONCAT(STR1:= ':',STR2:= sLastErrCode));
				fbLogger.mAddLine(sTextToSave := CONCAT(STR1:= 'Status NOK saved, StatusId- ', STR2:= LINT_TO_STRING(liLPartStatusId)));
				iCtr_PIM_PartsNOK := iCtr_PIM_PartsNOK +1;
			END_IF
			IF bLockAfterStatusSave THEN
				IF stPimInOut.sErrorCodePLC = '' THEN
					iConvTMP := nPIM_ErrorCodes.UnKnownLock;
					stPimInOut.sErrorCodePLC := INT_TO_STRING(iConvTMP);
				END_IF
				stPimInOut.bAlarmPLC :=  stPimInOut.bNonBlockingAlarm := FALSE;
				bSaveDefectRelation := stPimInOut.bWorkBlock_PLC := TRUE;				
			END_IF
		ELSE
			iCtr_StatusSaveError := iCtr_StatusSaveError + 1; 
			IF stSqlComandData.udiLEventId <> 0 THEN
				mSendCmdToPIM(sCmd := CONCAT(STR1:= 'StatusSaveError:', STR2:= UDINT_TO_STRING(stSqlComandData.udiLEventId)));
			ELSE
				mSendCmdToPIM(sCmd := 'StatusSaveError');
			END_IF
			IF bLastStatus THEN
				fbLogger.mAddLine(sTextToSave := 'Status OK Save error');
				iCtr_PIM_PartOK_SaveError := iCtr_PIM_PartOK_SaveError +1;
			ELSE
				fbLogger.mAddLine(sTextToSave := 'Status NOK Save error');
				iCtr_PIM_PartNOK_SaveError := iCtr_PIM_PartNOK_SaveError +1;
			END_IF
			IF bLockAfterStatusSave THEN
				IF stPimInOut.sErrorCodePLC = '' THEN
					iConvTMP := nPIM_ErrorCodes.UnKnownLock;
					stPimInOut.sErrorCodePLC := INT_TO_STRING(iConvTMP);
				END_IF
				bSaveDefectRelation := stPimInOut.bWorkBlock_PLC := TRUE;
			END_IF
		END_IF
		bPimCmdProcessing := bLockAfterStatusSave := bCmdSended := bInsertStatus := FALSE;		
		bReturnDataBusy := bReturnDataReserved_InsOperStat := FALSE;
	//	MEMSET(destAddr := ADR(stDBCmdData), n := SIZEOF(stDBCmdData), fillByte:= 0);		// Czyszczenie danych zapytania
	ELSIF NOT bPimCmdProcessing THEN
		bCmdSended := bInsertStatus := FALSE;
		bReturnDataBusy := bReturnDataReserved_InsOperStat := FALSE;
		IF bLockAfterStatusSave THEN
			IF stPimInOut.sErrorCodePLC = '' THEN
				iConvTMP := nPIM_ErrorCodes.UnKnownLock;
				stPimInOut.sErrorCodePLC := INT_TO_STRING(iConvTMP);
			END_IF
			stPimInOut.bAlarmPLC :=  stPimInOut.bNonBlockingAlarm := FALSE;
			stPimInOut.bWorkBlock_PLC := TRUE;		
			bLockAfterStatusSave := FALSE;		
		END_IF
	END_IF
ELSIF bLockAfterStatusSave AND stPimInOut.sErrorCodePLC <> '' THEN
//	{warning 'Wstawić sygnał zwrotny zapisu błędu do PIMu- zapis poprawny gdy nie są pobrane parametry z SQLa'}
	bLockAfterStatusSave := FALSE;
	stPimInOut.bAlarmPLC :=  stPimInOut.bNonBlockingAlarm := FALSE;
	stPimInOut.bWorkBlock_PLC := TRUE;	
END_IF


IF bSelPreviousStatus THEN 
	IF NOT bUpdateData THEN
		m_SqlSelLastOperationStatus(sCodeDM:= sLastDMCode, bProcessing => bPimCmdProcessing);
	END_IF
	IF stSqlComandData.bSQL_Done THEN
		IF  stSqlComandData.bSQL_OK THEN
			bPreviousOperationStatus := bPreviousOperationStatus;		
		END_IF
		bPimCmdProcessing := bCmdSended := bSelPreviousStatus := FALSE;
		bReturnDataBusy := bReturnDataReserved_SelLastOperStat := FALSE;
	ELSIF NOT bPimCmdProcessing THEN
		bCmdSended := bSelPreviousStatus := FALSE;
		bReturnDataBusy := bReturnDataReserved_SelLastOperStat := FALSE;		
	END_IF	
END_IF

IF bSelMachineParamsData THEN
	IF NOT bUpdateData THEN
		m_SqlSelMachineParamsData(diParamsId := 0, pParamsData:= 0, uiParamsDataSize := 0, bProcessing => bPimCmdProcessing);
	END_IF
	IF stSqlComandData.bSQL_Done THEN
		bPimCmdProcessing := bCmdSended := bSelMachineParamsData := FALSE;
		bReturnDataBusy := bReturnDataReserved_SelMachParams := FALSE;
	ELSIF NOT bPimCmdProcessing THEN
		bCmdSended := bSelMachineParamsData := FALSE;
		bReturnDataBusy := bReturnDataReserved_SelMachParams := FALSE;		
	END_IF
END_IF

IF bSelMachineParamsCRC THEN
	IF NOT bUpdateData THEN
		m_SqlSelMachineParamsCRC(liIdCompossedPart := 0, bProcessing => bPimCmdProcessing);
	END_IF
	IF stSqlComandData.bSQL_Done THEN
		IF stSqlComandData.bSQL_OK THEN
			diMachineParamsInsertId := diMachineParamsInsertId;
		END_IF
		bPimCmdProcessing := bCmdSended := bSelMachineParamsCRC := FALSE;
		bReturnDataBusy := bReturnDataReserved_SelMachParamsCRC := FALSE;
	ELSIF NOT bPimCmdProcessing THEN 
		bCmdSended := bSelMachineParamsCRC := FALSE;
		bReturnDataBusy := bReturnDataReserved_SelMachParamsCRC := FALSE;		
	END_IF
END_IF

IF bInsMachineParamsData THEN
	IF NOT bUpdateData THEN
		m_SqlInsMachineParamsData(pParamsData := 0, uiParamsDataSize := 0, wCrcSumOfParameters := 0, bProcessing => bPimCmdProcessing);
	END_IF
	IF stSqlComandData.bSQL_Done THEN
		IF stSqlComandData.bSQL_OK THEN
			diMachineParamsInsertId := diMachineParamsInsertId;
		END_IF
		bPimCmdProcessing := bCmdSended := bInsMachineParamsData := FALSE;
		bReturnDataBusy := bReturnDataReserved_InsMachParams := FALSE;
	ELSIF NOT bPimCmdProcessing THEN 
		bCmdSended := bInsMachineParamsData := FALSE;
		bReturnDataBusy := bReturnDataReserved_InsMachParams := FALSE;		
	END_IF
END_IF


ACT_UpdatePimOutput();
bUpdateData := FALSE;
END_ACTION

ACTION ACT_UpdatePimOutput:
(*
IF stPimInternal.sCmdPLC2PIM <> '' THEN
	stPimInOut.sCmdPLC2PIM := stPimInternal.sCmdPLC2PIM;	
	bCmdPlc2PimSended:= TRUE;
ELSIF sCmdPlc2PimBufer <> '' THEN
	stPimInternal.sCmdPLC2PIM := sCmdPlc2PimBufer; 
	bCmdPlc2PimSended:= TRUE;
ELSIF stPimInternal.sCmdPLC2PIM = '' THEN
	 stPimInOut.sCmdPLC2PIM := '';
END_IF
*)
END_ACTION

METHOD FB_init : BOOL
VAR_INPUT
	bInitRetains : BOOL; // if TRUE, the retain variables are initialized (warm start / cold start)
	bInCopyCode : BOOL;  // if TRUE, the instance afterwards gets moved into the copy code (online change)
	I_Mach: I_StationMachine;				// Interfejs do obsługi maszyn - pobranie danych z maszyny (głównie parametry pracy)
	I_Sql:	I_SQL_Core;		
END_VAR
I_Machine := I_Mach;
I_SqlCore := I_Sql;
END_METHOD

// Metoda zwraca strukturę do zapytania SQL uzupełnioną o dane z bloczka stanowiska
METHOD mGetStationData : stPIM_StationStatus
VAR_OUTPUT
	sCMD				: STRING;		// Zdarzenie jednostkowe/ rozkaz z PIMu np uaktualniono dane itp.
	bUserLogged			: BOOL;			// Użytkownik zalogowany
	bPIM_Active			: BOOL;			// Info o aktywności systemu PIM
	bTestMode			: BOOL;			// Aktywny tryb testowy
	bWorkPermittion		: BOOL;			// Informacja o zezwoleniu na pracę sumarycznie
	bWorkBlockPIM		: BOOL;			// Informacja o zezwoleniu na pracę z PIM
	bWorkBlockPLC		: BOOL;			// Informacja o zezwoleniu na pracę z PLC
	bConfirmation		: BOOL;			// Informacja o potwierdzeniu błędu
	bExternalMessage	: BOOL;			// Informacja o aktywnym komunikacie zewnętrznym
	nExtErrorClass		: nPIM_EventClasses;			// Informacja o aktywnym błędzie zewnętrznym
	bEventWaitInQueue	: BOOL;			// Info, że zdarzenie zewnętrzne czeka w kolejce
	nMachState			: nPIM_MachineStates;	// Aktualny status maszyny
	bOperInProgress		: BOOL;			// TRUE gdy operacja trwa
	bOperEnded			: BOOL;			// Impuls gdy operacja zakończona
	bOperStatus			: BOOL;			// Status ostatniej operacji
	nReworkSelected 	: nPIM_ReworkSelect;	// Operator wybrał Opcje reworku na tak lub nie
	nReoprtedNok 		: nPIM_ReportedNokSource;	// Operator zgłosił NOKa
END_VAR

mGetStationData:= stStationStatus;

sCMD := sCmdToSendToMachine;
sCmdToSendToMachine := '';
bUserLogged := fbTON_UserLogedDeleyed.Q;
bPIM_Active := stPimInOut.bPIMActive;
bWorkPermittion	:= bWorkPermitt;	
bWorkBlockPIM := stPimInOut.bWorkBlock_PIM;
bWorkBlockPLC := stPimInOut.bWorkBlock_PLC;
bConfirmation := stPimInOut.bConfirmEvent;
bTestMode := stPimInOut.bTestMode;
nExtErrorClass := nActExtErrorClass;
nMachState := nMachineState;
bEventWaitInQueue := iNextEventCodeEnum <> 0 AND bNextEventSource;

bOperInProgress := nMachineState = nPIM_MachineStates._4_OperationInProgress ;
bOperEnded := bOperationEnded OR nMachineState = nPIM_MachineStates._5_OperationEndedOK ;
bOperStatus := bLastStatus;
nReworkSelected:= nReworkMenuStatus;
nReoprtedNok := nReoprtedNokSource;
END_METHOD

METHOD PUBLIC mNewEvent : BOOL
VAR_INPUT
	iEventId:	INT;				// Kod błędu w postaci inta (do przekonwertowania)
	nEventType: nPIM_EventClasses;	// ROdzaj nowego zdarzenia
	tMessageTime: TIME:= T#3S;		// Czas na wyświetlenie wiadomości- ma znaczenie tylko dla wiadomości (po tym czasie lub po starcie nowej operacji wiadomość znika)
END_VAR
VAR
	sType: STRING;
END_VAR
// Zgłaszanie błędu zewnętrznego
IF nActIntErrorClass = nPIM_EventClasses.NoError THEN	// Jeśli aktualnienie ma aktywnego błędu dodaj jako podstawowy
	mNewEventCommon(iErrorEnum:= iEventId, nAlarmType := nEventType, tMessageTime := tMessageTime);
	nActExtErrorClass := nEventType;
ELSE	// Jeśli jest aktywny błąd wewnętrzny sprawdź co zrobić
	IF nEventType > nActIntErrorClass THEN	// Błąd zewnętrzny ważniejszy niż aktualny to
		IF nActIntErrorClass > nPIM_EventClasses.Message THEN 	// Jeśli aktywny wewnętrzny błąd ma priorytet wyższy niż wiadomość zamień błąd, a aktywny przenieś co pamięci 
			iNextEventCodeEnum := STRING_TO_INT(stPimInOut.sErrorCodePLC);
			nNextEeventType := nActIntErrorClass;
			bNextEventSource := FALSE;
			nActIntErrorClass := nPIM_EventClasses.NoError;
		ELSE	// Jeśli aktywna jest wiadomość tylko ją nadpisz
			nActIntErrorClass := nPIM_EventClasses.NoError;
			mNewEventCommon(iErrorEnum:= iEventId, nAlarmType := nEventType, tMessageTime := tMessageTime);
			nActExtErrorClass := nEventType;
		END_IF
	ELSE	// Błąd zewnętrzny ma niższy priorytet - dodanie nowego błędu do kolejki
		iNextEventCodeEnum := iEventId;
		nNextEeventType := nEventType;
		tNextEeventMessageTime := tMessageTime;
		bNextEventSource := TRUE;
	END_IF
END_IF

iCtr_NewEventCalls := iCtr_NewEventCalls+1;
IF nEventType = nPIM_EventClasses.Error THEN
	iCtr_NewEventCalls_ER := iCtr_NewEventCalls_ER +1;
ELSIF nEventType = nPIM_EventClasses.Alarm THEN
	iCtr_NewEventCalls_AL := iCtr_NewEventCalls_AL +1;
ELSE
	iCtr_NewEventCalls_Other := iCtr_NewEventCalls_Other +1;	
END_IF

// Logowanie danych
sType:= TO_STRING(nEventType);
fbFormatStr(sFormat := 'Nowy event zewnetrzny typ- %s, Id- %d',
	arg1 := F_STRINGEx(sType), 
	arg2 := F_INT(iEventId));  
fbLogger.mAddLine(sTextToSave := fbFormatStr.sOut );
mNewEvent := TRUE;

(*
IF NOT bInternalEventActive THEN	// Brak aktywnego alarmu lub aktywny alarm zewnętrzny (wtedy zamienia alarm)- dodaj alarm jako podstawowy
	mNewEventCommon(iErrorEnum:= iEventId, nAlarmType := nEventType, tMessageTime := tMessageTime);
	bExternalEventActive := nEventType = nPIM_EventClasses.Error OR nEventType = nPIM_EventClasses.Alarm;
	bExternalMessageActive := NOT bExternalEventActive;
	bInternalMessageActive := FALSE;		// Kasowanie wiadomości wewnętrznej (alarm ma wyższy priorytet
ELSE	// Alarm wewnętrzny jest już wyświetlany, dodaj alarm do kolejki
	
END_IF
*)
END_METHOD

// Kod wspólny dla zgłaszania błędów zewnętrznych i wewnętrznych
METHOD INTERNAL mNewEventCommon : BOOL
VAR_INPUT
	iErrorEnum:	INT;				// Kod błędu w postaci inta (do przekonwertowania)
	nAlarmType: nPIM_EventClasses;	// ROdzaj nowego zdarzenia
	tMessageTime: TIME:= T#3S;		// Czas na wyświetlenie wiadomości- ma znaczenie tylko dla wiadomości (po tym czasie lub po starcie nowej operacji wiadomość znika)
END_VAR
// Akcja z obsługą błędu - zmienne In_Out nie powinny być używane w metodach
// Określenie kodu alarmu
IF iErrorEnum <> 0 THEN		// Kod błędu podany przez Enum
	stPimInOut.sErrorCodePLC := INT_TO_STRING(iErrorEnum);
ELSE	// Brak kodu błędu -
	iConvTMP := nPIM_ErrorCodes.UnKnownLock;
	stPimInOut.sErrorCodePLC := INT_TO_STRING(iConvTMP);
END_IF		
bSaveDefectRelation R= NOT stPimInOut.bWorkBlock_PLC;

CASE nAlarmType OF 
	nPIM_EventClasses.Error:		// Błąd związany z częścią - trzeba bezwzględnie zapisać status i wtedy wystawić odpowiednie bity (Chyba, że status został zapisany
		IF bSaveDefectRelation THEN
			IF stPimInOut.sStatusNokAndErrorID = CONCAT(STR1:= LINT_TO_STRING(liLPartStatusId), STR2:= CONCAT(STR1:= ':',STR2:= stPimInOut.sErrorCodePLC)) THEN
				stPimInOut.sStatusNokAndErrorID := '';
				fbTON_WriteErrorCode2Status.IN:= TRUE;	
			ELSE
				stPimInOut.sStatusNokAndErrorID := CONCAT(STR1:= LINT_TO_STRING(liLPartStatusId), STR2:= CONCAT(STR1:= ':',STR2:= stPimInOut.sErrorCodePLC));
			END_IF
	//		m_SqlInsDefectRelation(sErrCode := stPimInternal.sKomunikatBladPlc);
		ELSE
			m_SqlSelInsStatus(bStatus := FALSE, sErrCode := stPimInOut.sErrorCodePLC, bSustein := TRUE);	
			fbLogger.mAddLine(sTextToSave := CONCAT(STR1:= 'Relation added to the last StatusId- ', STR2:= LINT_TO_STRING(liLPartStatusId)));
			bStatusSaveTriggered := bLockAfterStatusSave := TRUE;	
		END_IF
	//	m_SqlSelInsStatus(bStatus := FALSE, sErrCode := stPimInOut.sErrorCodePLC, bSustein := TRUE);
	//	bStatusSaveTriggered := bLockAfterStatusSave := TRUE;	
		iCtr_Errors:= iCtr_Errors + 1; 
		iCtr_NewComEventCalls_ER := iCtr_NewComEventCalls_ER +1;
	nPIM_EventClasses.Alarm:
		stPimInOut.bAlarmPLC := NOT stPimInOut.bWorkBlock_PLC;	// Jeśli jest już aktywne blokowanie, nie aktywuj alarmu tylko zmień kod błędu
		stPimInOut.bNonBlockingAlarm := FALSE;
		m_SqlInsAdditionalError(sErrCode:= stPimInOut.sErrorCodePLC);
		iCtr_NewComEventCalls_AL := iCtr_NewComEventCalls_AL +1;
		
	nPIM_EventClasses.AlarmAutoConfirm:
		stPimInOut.bNonBlockingAlarm := stPimInOut.bAlarmPLC := NOT stPimInOut.bWorkBlock_PLC;
		m_SqlInsAdditionalError(sErrCode:= stPimInOut.sErrorCodePLC);
		iCtr_NewComEventCalls_Other := iCtr_NewComEventCalls_Other +1;

	nPIM_EventClasses.Message:
		stPimInOut.bNonBlockingAlarm := stPimInOut.bAlarmPLC := NOT stPimInOut.bWorkBlock_PLC;
		fbTON_MessageTimer(IN:= TRUE, PT := tMessageTime);
		iCtr_NewComEventCalls_Other := iCtr_NewComEventCalls_Other +1;
END_CASE	
ACT_UpdatePimOutput();
mNewEventCommon := TRUE;
END_METHOD

METHOD INTERNAL mNewlnternalEvent : BOOL
VAR_INPUT
	nInputErrorID:	nPIM_ErrorCodes;	// Kod błędu w postaci inta (do przekonwertowania)
	nEventType: nPIM_EventClasses;	// ROdzaj nowego zdarzenia
	tMessageTime: TIME:= T#3S;		// Czas na wyświetlenie wiadomości- ma znaczenie tylko dla wiadomości (po tym czasie lub po starcie nowej operacji wiadomość znika)
END_VAR
VAR
	sType: STRING;
END_VAR
// Jeśli aktualnie brak błędu lub błąd o niższym priorytecie zamień błędy, jeśli nie zapisz na przyszłość
IF nActExtErrorClass = nPIM_EventClasses.NoError THEN
	mNewEventCommon(iErrorEnum:= nInputErrorID, nAlarmType := nEventType, tMessageTime := tMessageTime);
	nActIntErrorClass := nEventType;
ELSIF nEventType > nActExtErrorClass AND nActExtErrorClass > nPIM_EventClasses.Message THEN	// Alarm wewn. ma wyższy priorytet - przesuń aktywny alarm do kolejki
	iNextEventCodeEnum := STRING_TO_INT(stPimInOut.sErrorCodePLC);
	nNextEeventType := nActExtErrorClass;
	bNextEventSource := TRUE;
	nActExtErrorClass := nPIM_EventClasses.NoError;

ELSE
	iNextEventCodeEnum := nInputErrorID;
	nNextEeventType := nEventType;
	tNextEeventMessageTime := tMessageTime;
	bNextEventSource := FALSE;
END_IF

iCtr_NewIntEventCalls := iCtr_NewIntEventCalls + 1;
nErrorID := nInputErrorID;
sType := TO_STRING(nEventType);
fbFormatStr(sFormat := 'Nowy event wewnetrzny typ- %s, Id- %d',arg1 := F_STRINGEx(sType), arg2 := F_INT(nErrorID));  
fbLogger.mAddLine(sTextToSave := fbFormatStr.sOut );
iWorkStep := 99;
END_METHOD

METHOD mNewServiceMessage : BOOL
VAR_INPUT
	sMessage: STRING(255);			// Wiadomośćdo wyświetlenia
	tMessageTime: TIME:= T#3S;		// Czas na wyświetlenie wiadomości- ma znaczenie tylko dla wiadomości (po tym czasie lub po starcie nowej operacji wiadomość znika)	
END_VAR
stPimInOut.sPlcServiceMessage := sMessage;
IF tMessageTime > T#100MS THEN
	fbTON_ServiceMessageTimer(IN:= FALSE);	
	fbTON_ServiceMessageTimer(IN:= TRUE, PT:= tMessageTime);	
END_IF
END_METHOD

METHOD INTERNAL mSendCmdToPIM : BOOL
VAR_INPUT
	sCmd: STRING;
END_VAR
IF stPimInOut.sCmdPLC2PIM = '' THEN		// Cmd Empty
	stPimInOut.sCmdPLC2PIM := CONCAT(STR1:= sCmd, STR2:= ';');
ELSE	// Not empty - check if cmd isnt sended
	IF NOT bCmdPlc2PimSended THEN
		IF RIGHT(STR:= stPimInOut.sCmdPLC2PIM, SIZE:= 1) <> ';' THEN		// Separator are not present
			stPimInOut.sCmdPLC2PIM := CONCAT(STR1:= stPimInOut.sCmdPLC2PIM, STR2:= ';');	
		END_IF
		stPimInOut.sCmdPLC2PIM := CONCAT(STR1:= sCmd, STR2:= 'sCmd');
		stPimInOut.sCmdPLC2PIM := CONCAT(STR1:= stPimInOut.sCmdPLC2PIM, STR2:= ';');
	ELSE		// Write cmd in bufer		
		IF sCmdPlc2PimBufer = '' THEN		// Cmd Empty
			sCmdPlc2PimBufer := CONCAT(STR1:= sCmd, STR2:= ';');
		ELSE	// Not empty
			IF RIGHT(STR:= sCmdPlc2PimBufer, SIZE:= 1) <> ';' THEN		// Separator are not present
				sCmdPlc2PimBufer := CONCAT(STR1:= sCmdPlc2PimBufer, STR2:= ';');	
			END_IF
			sCmdPlc2PimBufer := CONCAT(STR1:= sCmd, STR2:= 'sCmd');
			sCmdPlc2PimBufer := CONCAT(STR1:= sCmdPlc2PimBufer, STR2:= ';');
		END_IF
	END_IF
END_IF
mSendCmdToPIM := TRUE;
END_METHOD

// Masyzna zgłasza chęć przejścia do nowego stanu/kroku - pim wydaje zezwolenie na zmianę stanu dla poszczególnych kroków bazując na stanie z systemu PIM
METHOD mSetNewMachineState : BOOL
VAR_INPUT
	nMachineNewState: nPIM_MachineStates;		// Nowy stan maszyny
END_VAR

// Obsługa kodu tylko gdy stan się zmienia 
IF nMachineNewState <> nMachineState THEN
	//	**************************************************** Określenie zezwolenia **************************************************** 
	CASE nMachineNewState OF	// Wydanie zezwolenia na przejście do kolejnego kroku 
		
		nPIM_MachineStates._3_NewOperationStarted:		// Zezwolenie na start nowej operacji	
			mSetNewMachineState := bWorkPermitt; 
			
		nPIM_MachineStates._6_ReturningToBaseState:		// Zezwolenie na zwolnienie części (np gdy operator się wylogował lub koniec zlecenia, pełny box itp... (Future Reference)
			mSetNewMachineState := TRUE;
			
		nPIM_MachineStates._9_ResetInProgress:			// Maszyna w oczekiwaniu na potwierdzenie błędu - powinna wysłać numer błędu- sprawdź czy wyświetlany jest błąd
			IF nActExtErrorClass <> nPIM_EventClasses.NoError THEN	// Jeśli jest aktywny błąd lub wiadomość zewnętrzna to wszystko OK- można wysłać sygnał resetu do maszyny.
				mSetNewMachineState := stPimInOut.bConfirmEvent;	// OR bPIM_Working;	
			ELSIF iNextEventCodeEnum = 0 THEN	// Jeśli błędu nie ma w kolejce a maszyna jest w błędzie - błąd w działaniu maszyny
				IF nActIntErrorClass = nPIM_EventClasses.NoError THEN
					mNewEvent(iEventId:= nPIM_ErrorCodes.MachErrorWhenNoErrorCode, nEventType := nPIM_EventClasses.Alarm, tMessageTime := T#0S);
				ELSE
					iNextEventCodeEnum := nPIM_ErrorCodes.MachErrorWhenNoErrorCode;
					nNextEeventType := nPIM_EventClasses.Alarm;
					tNextEeventMessageTime := T#0S;
					bNextEventSource := TRUE;
				END_IF
				nMachineState := nPIM_MachineStates._8_WaitForReset;		// Zaktualizowanie stanu maszyny w PIMie
			END_IF
			stPimInOut.bConfirmEvent R= mSetNewMachineState;
	ELSE	// W innych przypadkach zezwalaj - do potencjalnego późniejszego rozszerzenia
		mSetNewMachineState := TRUE;
	END_CASE
	
	
	
//	************************************ Jeśli jest zezwolenie zaktualizuj stan w bloczku PIM ****************************************
	IF mSetNewMachineState THEN		// Jeśli wydano zezwolenie na przejście do kolejnego kroku zaktualizuj stan maszyny w PIMie
		
		IF nMachineNewState = nPIM_MachineStates._3_NewOperationStarted THEN
			// Można też sprawdzić zapis poprzedniego statusu
			bNewOperationStartedMethod := TRUE;
		ELSIF nMachineNewState = nPIM_MachineStates._5_OperationEndedOK THEN
			m_SqlSelInsStatus(bStatus := TRUE, sErrCode := '', bSustein := TRUE);
			bNewOperationEndedOKMethod := bStatusSaveTriggered := TRUE;		
			iCtr_OperEndedOK_Method := iCtr_OperEndedOK_Method + 1;
		ELSIF nMachineNewState = nPIM_MachineStates._7_ErrorOccurr THEN
			// W przypadku błędu blok FB maszyny powinien najpierw zgłosić błąd, potem zaraportować zmianę kroku na np. ErrorOccurr
			bOperationEndedErrorMethod := TRUE;		
		END_IF
		
		// Jeśli reset błędu/alarmu w maszynie zakończony porawnie wyzeruj zmienne od alarmowania
		IF nMachineState = nPIM_MachineStates._9_ResetInProgress THEN
			stPimInOut.bConfirmEvent := FALSE;		// Podejrzenie, że w czasie resetu jest kilka razy wysyłany ten sam kod błędu (pętla nieskończona gdy sygnał ustawiony i błąd w FB_Maszyny)
			IF (nMachineNewState = nPIM_MachineStates._0_Standby_NotReady OR nMachineNewState = nPIM_MachineStates._0_Initialization)  THEN // Reset w maszynie zakończony poprawnie
				IF nActExtErrorClass <> nPIM_EventClasses.NoError THEN		// Wszystko OK maszyna zgłosiła uprzednio błąd 
					fbLogger.mAddLine(sTextToSave := CONCAT(STR1:= 'ResetExtError- ', STR2:= stPimInOut.sErrorCodePLC ) );
					stPimInOut.bNonBlockingAlarm := stPimInOut.bAlarmPLC := stPimInOut.bWorkBlock_PLC := FALSE;
					stPimInOut.sErrorCodePLC := '';
					nActExtErrorClass := nPIM_EventClasses.NoError;
					bSaveDefectRelation := stPimInOut.bConfirmEvent	:= FALSE;		
				ELSIF nActIntErrorClass = nPIM_EventClasses.NoError THEN	// Maszyna wykonała reset pomimo braku aktywnego alarmu - Coś jest nie tak ale wygaś okno alarmowe
					fbLogger.mAddLine(sTextToSave := CONCAT(STR1:= 'EmergErrReset- ', STR2:= stPimInOut.sErrorCodePLC ) );
					stPimInOut.bNonBlockingAlarm := stPimInOut.bAlarmPLC := stPimInOut.bWorkBlock_PLC := FALSE;
					stPimInOut.sErrorCodePLC := '';
					bSaveDefectRelation := stPimInOut.bConfirmEvent	:= FALSE;		
				END_IF
			//ELSIF nMachineState = nPIM_MachineStates._7_ErrorOccurr THEN
			
			//	mNewlnternalEvent(nInputErrorID:= nPIM_ErrorCodes.ProgramError, nEventType := nPIM_EventClasses.Error, tMessageTime := T#0S);
			//	fbLogger.mAddLine(sTextToSave := CONCAT(STR1:= 'InvalidStateAfterReset- ', STR2:= INT_TO_STRING(nMachineNewState) ) );	
			END_IF
		END_IF 
			
		nMachineState := nMachineNewState;	
	END_IF
ELSIF nMachineNewState = nPIM_MachineStates._2_ReadyForNewOperation AND nActExtErrorClass > nPIM_EventClasses.AlarmAutoConfirm THEN
	fbLogger.mAddLine(sTextToSave := CONCAT(STR1:= 'MachineResetWithoutAck, error-', STR2:= stPimInOut.sErrorCodePLC ) );
	stPimInOut.bNonBlockingAlarm := stPimInOut.bAlarmPLC := stPimInOut.bWorkBlock_PLC := FALSE;
	stPimInOut.sErrorCodePLC := '';		
	nActExtErrorClass := nPIM_EventClasses.NoError;
	stPimInOut.bConfirmEvent	:= FALSE;	
END_IF
ACT_UpdatePimOutput();
END_METHOD

END_FUNCTION_BLOCK

// PIM/POUs/fbPIM_UserLogin
FUNCTION_BLOCK fbPIM_UserLogin
VAR_INPUT
	tLogoutTime: TIME:= T#5M;	// Czas do auto wylogowania, gdy T#0s automatyczne wylogowanie wyłączone
END_VAR
VAR_OUTPUT
	nUserRole:nSQL_UserRoles;
	bUserLogged:BOOL;
	sUserName:STRING;
	bSqlDone : BOOL;
	bSqlError : BOOL;
END_VAR
VAR
	I_SqlCore: I_SQL_Core;
	sScanedId : STRING(50):= '';
	stSqlComandData: stSQL_ClientNode;
	fbTonSelect : TON;
	sCodeNumber:STRING(50);
    sCmd : STRING (255); 
    stRetDataUserRole:stSQL_RetDataUserRole;	
	iRepeatExecutionCtr: INT;
	sEventText: STRING;
	bZezwolenie: BOOL;
	bSQLQueryActive: BOOL;
	nRecordsLineStation: UDINT;
	bSelectRole: BOOL;
	fbTON_Logout: TON;
	bPermissionGranted: BOOL;
	fbFTRIG_Logout: F_TRIG;
	asLogHistory:ARRAY [1..20] OF STRING;
	bCmdSended: BOOL;
END_VAR

IF  LEN(sScanedId) > 2 THEN	// Zeskonowano nową kartę
	IF sScanedId = 'yyXAzyD6ZLy' OR sScanedId = '4DgQLtbNKPJ' OR sScanedId = 'u9r6EnxFXqm' OR sScanedId = 'has10mas10' THEN
		// Reakcja awaryjna w przypadku gdy normalne karty nie działają, karta nadrzędna - nie sprawdza uprawnień w bazie danych
		nUserRole := nSQL_UserRoles.AdminUser;
		sUserName := 'Admin User';
		bSqlDone := bPermissionGranted := bUserLogged := TRUE;
		MEMMOVE(srcAddr := ADR(asLogHistory[1]), destAddr := ADR(asLogHistory[2]), n := 19*SIZEOF(asLogHistory[1]));
		asLogHistory[1] := CONCAT(STR1:= DT_TO_STRING(GVL_Aircom.stAC_DT_Data.dtActualDate), STR2 := CONCAT(STR1:= '- ', STR2:= sUserName)) ;
	ELSIF sScanedId = '555444' THEN
		// Reakcja awaryjna w przypadku gdy normalne karty nie działają, karta nadrzędna - nie sprawdza uprawnień w bazie danych
		nUserRole := nSQL_UserRoles.Maintenance;
		sUserName := 'Maintenance User';
		bSqlDone := bPermissionGranted := bUserLogged := TRUE;
		MEMMOVE(srcAddr := ADR(asLogHistory[1]), destAddr := ADR(asLogHistory[2]), n := 19*SIZEOF(asLogHistory[1]));
		asLogHistory[1] := CONCAT(STR1:= DT_TO_STRING(GVL_Aircom.stAC_DT_Data.dtActualDate), STR2 := CONCAT(STR1:= '- ', STR2:= sUserName)) ;
	ELSE	// Gdy baza danych działa zapytaj o uprawnienia
		// Dane do zapytania
		sCodeNumber := MID(STR:= sScanedId,POS:= 4, LEN:= LEN(sScanedId)-3);		// Usunięcie prefixu 'ID_'
		bSqlDone := bSqlError := FALSE;
		IF LEN(sCodeNumber) >= 1 THEN
			stSqlComandData.nCmdState:= nSQL_CmdExecState.New;
			stSqlComandData.nCmdType:=nSQL_CmdTypes.SelUserRole;
			stSqlComandData.bWaitForDataReturn:=TRUE;
			sCmd := CONCAT('SELECT Role, FirstName, LastName FROM ProductionUser WHERE Active=1 AND CodeNumber = $'',sCodeNumber); 
			sCmd := CONCAT(sCmd,'$''); 
			stSqlComandData.sCmdExpression := sCmd;
//			stSqlComandData.stCmdData.sName0 := sCodeNumber; 
			stSqlComandData.pReturnedData := ADR(stRetDataUserRole);
			stSqlComandData.uiReturnedDataSize := SIZEOF(stRetDataUserRole);
			stSqlComandData.bSQL_OK := stSqlComandData.bSQL_Done := FALSE;
			bPermissionGranted := bUserLogged := FALSE;
			IF I_SqlCore <> 0 AND_THEN I_SqlCore.mAddCmdToQueue(ADR(stSqlComandData)) THEN		// Próba dodania komendy do kolejki
				bCmdSended := TRUE;		// Zajęcie struktury danych
				MEMSET(destAddr := ADR(stRetDataUserRole), n := SIZEOF(stRetDataUserRole), fillByte:= 0);		// Czyszczenie danych 
			ELSE
				bCmdSended := FALSE;
				bSqlDone := bSqlError := TRUE;
			END_IF
		END_IF	
	END_IF
	sScanedId := '';
ELSE
	sScanedId := '';	
END_IF

IF bCmdSended AND stSqlComandData.bSQL_Done THEN
	bSqlDone := TRUE;
	IF stSqlComandData.bSQL_OK THEN
		IF stRetDataUserRole.Role = '' THEN
			nUserRole := nSQL_UserRoles.NONE;
			bPermissionGranted := FALSE;
		ELSIF stRetDataUserRole.Role = 'Operator' THEN
			nUserRole := nSQL_UserRoles.Operator;
			bPermissionGranted := FALSE;
		ELSIF stRetDataUserRole.Role = 'Quality' THEN
			nUserRole := nSQL_UserRoles.Quality;
			bPermissionGranted := FALSE;
		ELSIF stRetDataUserRole.Role = 'RDChem' THEN
			nUserRole := nSQL_UserRoles.RDChem;
			bPermissionGranted := FALSE;	
		ELSIF stRetDataUserRole.Role = 'Trainer' THEN
			nUserRole := nSQL_UserRoles.Trainer;
			bPermissionGranted := FALSE;	
		ELSIF stRetDataUserRole.Role = 'Maintenance' THEN
			nUserRole := nSQL_UserRoles.Maintenance;
			bPermissionGranted := TRUE;
		ELSIF stRetDataUserRole.Role = 'LineLeader' THEN
			nUserRole := nSQL_UserRoles.LineLeader;
			bPermissionGranted := TRUE;
		ELSIF stRetDataUserRole.Role = 'ShiftLeader' THEN
			nUserRole := nSQL_UserRoles.ShiftLeader;
			bPermissionGranted := TRUE;
		ELSIF stRetDataUserRole.Role = 'Supervisor' THEN
			nUserRole := nSQL_UserRoles.Supervisor;
			bPermissionGranted := TRUE;
		ELSIF stRetDataUserRole.Role = 'RD' THEN
			nUserRole := nSQL_UserRoles.RD;
			bPermissionGranted := TRUE;
		ELSIF stRetDataUserRole.Role = 'Engineering' THEN
			nUserRole := nSQL_UserRoles.Engineering;
			bPermissionGranted := TRUE;
		ELSIF stRetDataUserRole.Role = 'Admin' THEN
			nUserRole := nSQL_UserRoles.AdminUser;
			bPermissionGranted := TRUE;
		ELSE
			nUserRole := nSQL_UserRoles.Unspecified;
			bPermissionGranted := FALSE;
		END_IF
		IF nUserRole <> nSQL_UserRoles.NONE THEN
			sUserName := CONCAT(STR1:=stRetDataUserRole.FirstName, STR2:= CONCAT(STR1:= '  ', STR2:= stRetDataUserRole.LastName));
			bUserLogged := TRUE;
			MEMMOVE(srcAddr := ADR(asLogHistory[1]), destAddr := ADR(asLogHistory[2]), n := 19*SIZEOF(asLogHistory[1]));
			asLogHistory[1] := CONCAT(STR1:= DT_TO_STRING(GVL_Aircom.stAC_DT_Data.dtActualDate), STR2 := CONCAT(STR1:= '- ', STR2:= sUserName)) ;
		END_IF
		GVL_Aircom.nUserRole := nUserRole;
		GVL_Aircom.sUserName := sUserName;
		GVL_Aircom.bUserLogged := bUserLogged;
		GVL_Aircom.bPermissionGranted := bPermissionGranted;
		bSqlDone := TRUE;
		bSqlError := FALSE;
	ELSE
		nUserRole := nSQL_UserRoles.Unspecified;
		bPermissionGranted := FALSE;
		bSqlDone := bSqlError := TRUE;
	END_IF
	bCmdSended := FALSE;	
END_IF
fbFTRIG_Logout(CLK:= bUserLogged);
IF tLogoutTime > T#0S THEN
	fbTON_Logout(IN:=bUserLogged,PT:=tLogoutTime);
ELSE
	fbTON_Logout(IN:=FALSE,PT:=T#1H);
END_IF
IF fbTON_Logout.Q OR fbFTRIG_Logout.Q THEN
	GVL_Aircom.nUserRole := nUserRole := nSQL_UserRoles.NONE;
	GVL_Aircom.sUserName := sUserName := sUserName:= 'none';
	GVL_Aircom.bUserLogged := bUserLogged := FALSE;
	GVL_Aircom.bPermissionGranted := bPermissionGranted := FALSE;
END_IF

METHOD FB_init : BOOL
VAR_INPUT
	bInitRetains : BOOL; // if TRUE, the retain variables are initialized (warm start / cold start)
	bInCopyCode : BOOL;  // if TRUE, the instance afterwards gets moved into the copy code (online change)
	I_Sql: I_SQL_Core;
END_VAR
I_SqlCore := I_Sql;
END_METHOD

END_FUNCTION_BLOCK

// ProdLineMachines/AssemblyPost/fbAssemblyPost
FUNCTION_BLOCK PUBLIC fbAssemblyPost IMPLEMENTS I_StationMachine
VAR_IN_OUT
	stWorkParams		: stAssemblyPost_Settings;		// Fixture settings and parameters
END_VAR
VAR_INPUT
	bPartSensor			: BOOL;				// When part in fixation
	bPartSensorInvert	: BOOL;				// Invert logic of compressor sensor input
	tFilterTime			: TIME:= T#350MS;	// Input signal filtration time
END_VAR
VAR_OUTPUT
	bPartLock_Q			: BOOL;
	nError:nAssemblyPost_ErrorList;			// Active error
END_VAR
VAR
	I_PimSystem			: I_PIM;		// PIM Interface
	pParamsStruct	: POINTER TO BYTE;		// 	Wskaźnik do parametrów pracy maszyny
	uiParamsSize	: UINT;						// 	Rozmiar struktury parametrów pracy maszyny [bajty]
	fbPartFiltered: fbBinaryFilter;	
	iWorkStep: INT;
	fbTON_PartInFixture, fbTON_PartOutFixture: TON;
	iPartRemToFast, ipartPutToFast, iPartsMissed: INT;		// Liczniki potencjalnych błędów
	iPartPutToFastMem, iPartRemToFastMem, iPartsMissedMem: INT;	// Liczniki błędów z poprzedniej zmiany
	
	bUserLogged: BOOL;
	bPIM_Active: BOOL;
	stStationData: stPIM_StationStatus;

END_VAR

// Filtrowanie sygnału obeności kompresora w kowadle - sygnał ustawiany gdy jest sygnał z czujnika jest przez tInputFlterTime, resetowany podobnie
fbPartFiltered(In := bPartSensor XOR bPartSensorInvert, tON := tFilterTime, tOFF := tFilterTime/2);

stStationData:= I_PimSystem.mGetStationData(bUserLogged => bUserLogged,
		bPIM_Active => bPIM_Active);
pParamsStruct := ADR(stWorkParams);
uiParamsSize := SIZEOF(stWorkParams);

IF fbPartFiltered.FTrig AND iWorkStep <> 10 THEN
	iPartsMissed := iPartsMissed + 1;
END_IF
CASE iWorkStep OF 
	0:	// Inicjalizacja
		I_PimSystem.mSetNewMachineState(nPIM_MachineStates._0_Initialization);
		iWorkStep := 1;
		
	1:	// 
		I_PimSystem.mSetNewMachineState(nPIM_MachineStates._0_Standby_NotReady);
		fbTON_PartOutFixture(IN:= FALSE);
		iWorkStep := 5;
		
	5:	// Krok spoczynkowy - oczekiwanie na nową operację
		I_PimSystem.mSetNewMachineState(nPIM_MachineStates._2_ReadyForNewOperation);
		bPartLock_Q := NOT bUserLogged;
		IF fbPartFiltered.Q THEN
			IF I_PimSystem.mSetNewMachineState(nPIM_MachineStates._3_NewOperationStarted) THEN
				fbTON_PartInFixture(IN:= FALSE);
				IF fbTON_PartOutFixture.Q THEN			// Część włożona po wymaganym czasie
					bPartLock_Q := TRUE;
					iWorkStep := 10;
				ELSE
					IF stWorkParams.bMonitorOFF_Time THEN	// Czy kontrola czasu OFF włączona?
						mNewEvent(nEventClass:= nPIM_EventClasses.Error, nEvent := nAssemblyPost_ErrorList.PartInsertedToFast);
					ELSE 
						ipartPutToFast := ipartPutToFast +1;
						iWorkStep := 10;
					END_IF					
				END_IF			
			END_IF		
		END_IF
				
	10:	// Trwa montaż...
		I_PimSystem.mSetNewMachineState(nPIM_MachineStates._4_OperationInProgress);
		IF NOT fbPartFiltered.Q THEN
			IF NOT fbTON_PartInFixture.Q THEN			// Część wyciągnięta zbyt szybko
				IF stWorkParams.bMonitorON_Time THEN	// Czy kontrola czasu ON włączona?
					mNewEvent(nEventClass:= nPIM_EventClasses.Error, nEvent := nAssemblyPost_ErrorList.PartRemovedToFast);
				ELSE 
					iPartRemToFast := iPartRemToFast +1;
					iWorkStep := 15;
				END_IF
			ELSE
				iWorkStep := 15;
			END_IF
		END_IF
		
	15:	// Operacja zakończOna OK
		I_PimSystem.mSetNewMachineState(nPIM_MachineStates._5_OperationEndedOK);
		iWorkStep := 20;
		
	20: // Powrót do stanu początkowego
		IF I_PimSystem.mSetNewMachineState(nPIM_MachineStates._6_ReturningToBaseState) THEN
			bPartLock_Q := FALSE;
			iWorkStep := 1;
		END_IF

	90:	// Blokowanie stanowiska, 90 - zapis statusu + kod błędu, 91 - zapis dodatkowego błędu
		bPartLock_Q := TRUE;
		I_PimSystem.mSetNewMachineState(nPIM_MachineStates._8_WaitForReset);
		iWorkStep := 91;
		
	91:	// Oczekiwanie na pozytywne zakończenie zapisu statusu NOK do DB
		IF I_PimSystem.mSetNewMachineState(nPIM_MachineStates._9_ResetInProgress) THEN
			iWorkStep := 95;
		END_IF
		
	95:	// Reset
		bPartLock_Q := FALSE;
		iWorkStep := 1;
END_CASE

// Statistics
IF GVL_Aircom.stAC_DT_Data.bNew_Shift THEN
	iPartPutToFastMem := ipartPutToFast;
	iPartRemToFastMem := iPartRemToFast;
	iPartsMissedMem := iPartsMissed;
	ipartPutToFast := iPartRemToFast := 0;
END_IF

fbTON_PartOutFixture(IN:=  NOT fbPartFiltered.Q, PT:= REAL_TO_TIME(1000*stWorkParams.rRequiredTimeOFF));
fbTON_PartInFixture(IN:= fbPartFiltered.Q, PT:= REAL_TO_TIME(1000*stWorkParams.rRequiredTimeON));

METHOD FB_init : BOOL
VAR_INPUT
	bInitRetains : BOOL; // if TRUE, the retain variables are initialized (warm start / cold start)
	bInCopyCode : BOOL;  // if TRUE, the instance afterwards gets moved into the copy code (online change)
	I_Pim	: I_PIM;		// Interfejs do bloku PIM
END_VAR
I_PimSystem := I_Pim;
END_METHOD

(* Metoda TRUE kiedy dane wyjściowe są ok, jeśli nie FALSE (jeśli not bBusy i FALSE to błąd odczytu) *)
METHOD mGetParamsData : BOOL
VAR_INPUT
	bTestParams:	BOOL;	// Jeśli TRUE metoda okresla czy ma dostęp do parametrów, jeśli tak zwraca TRUE, jeśli nie FALSE
END_VAR
VAR_OUTPUT
	bBusy	: BOOL;										//	Maszyna odświeża dane
	pMachineParametersStruct	: POINTER TO BYTE;		// 	Wskaźnik do parametrów pracy maszyny
	uiMachineParametersSize	: UINT;						// 	Rozmiar struktury parametrów pracy maszyny [bajty]
	wActualCRC16SumInMachine	: WORD;					//	Aktualna suma CRC16 obliczona z parametrów
END_VAR
pMachineParametersStruct := pParamsStruct;
uiMachineParametersSize := uiParamsSize;
wActualCRC16SumInMachine := F_DATA_TO_CRC16_CCITT(pData := pMachineParametersStruct, cbData := uiMachineParametersSize, crc := 16#0000);
bBusy := FALSE;
mGetParamsData := TRUE;
END_METHOD

METHOD INTERNAL mNewEvent : BOOL
VAR_INPUT
	nEventClass:nPIM_EventClasses;
	nEvent: nAssemblyPost_ErrorList;
END_VAR
IF nEventClass = nPIM_EventClasses.AlarmAutoConfirm OR nEventClass = nPIM_EventClasses.Message THEN		// Alarm nieblokadowy
	I_PimSystem.mSetNewMachineState(nPIM_MachineStates._0_Initialization);
	iWorkStep := 90;
ELSE
	I_PimSystem.mSetNewMachineState(nPIM_MachineStates._7_ErrorOccurr);
	I_PimSystem.mNewEvent(iEventId := nEvent, nEventType := nEventClass, tMessageTime := T#0S);
	iWorkStep := 90;
END_IF
nError := nEvent;
END_METHOD

END_FUNCTION_BLOCK

// ProdLineMachines/S02_ManometerTubeAssy/V1/fbManometerTubeAssy_V1
FUNCTION_BLOCK fbManometerTubeAssy_V1 IMPLEMENTS I_StationMachine
VAR_IN_OUT
	stInOuts: stManometerTubeAssy_InOuts;
END_VAR
VAR_INPUT
	tDeltaDwuStart:TIME:= T#200MS;
END_VAR
VAR_OUTPUT
	nError:nManometerTubeAssy_ErrorCodes;
END_VAR
VAR
	I_PimSystem			: I_PIM;
	fb2Start: fb2HandStartBasic;
	udiOperationsOK_Qty: UDINT;
	iWorkStep: INT;
	fbTON_StepTimeout: TON;
	
	bServiceReset: BOOL;
END_VAR

fb2Start(stInOutsData:= stInOuts.st2HandStartIO, tDeltaDwuStart := T#250MS);

//  Błędy monitorowane stale (bezpieczeństwo)
IF NOT stInOuts.st2HandStartIO.bEmergButton_NC AND iWorkStep <> 95 AND nError <> nManometerTubeAssy_ErrorCodes.SafetySystemNotArmed THEN
	stInOuts.bPressValve_Q := FALSE;
	mNewEvent(nEvent:=nManometerTubeAssy_ErrorCodes.SafetySystemNotArmed , nEventClass := nPIM_EventClasses.Error);
END_IF

CASE iWorkStep OF 
	0:	// Inicjalizacja
		I_PimSystem.mSetNewMachineState(nPIM_MachineStates._0_Initialization);
		stInOuts.bPressValve_Q := FALSE;
		iWorkStep := 1;
		
	1:	// Init
		I_PimSystem.mSetNewMachineState(nPIM_MachineStates._0_Standby_NotReady);
		iWorkStep := 5;
	
	5:	// Krok spoczynkowy - oczekiwanie na nową operację
		I_PimSystem.mSetNewMachineState(nPIM_MachineStates._2_ReadyForNewOperation);
		IF fb2Start.bStartSig AND stInOuts.bPressHomePos AND stInOuts.bHandleWorkPos  THEN
			IF I_PimSystem.mSetNewMachineState(nPIM_MachineStates._3_NewOperationStarted) THEN 
				iWorkStep := 10;
				fbTON_StepTimeout(IN:= FALSE);
			END_IF
		END_IF
		
	10:	// Nowa operacja rozpoczęta - ustawienie sygnałów
		fbTON_StepTimeout(IN:= TRUE, PT:= T#500MS);
		IF fb2Start.bStartSig THEN
			stInOuts.bPressValve_Q := TRUE;
			IF NOT stInOuts.bPressHomePos THEN	// Jest ruch siłownika
				iWorkStep := 15;
			ELSIF fbTON_StepTimeout.Q THEN
				stInOuts.bPressValve_Q := TRUE;
				mNewEvent(nEventClass:= nPIM_EventClasses.Alarm, nEvent:= nManometerTubeAssy_ErrorCodes.NoMachineReactionOnStartSig);
			END_IF
		ELSE
			stInOuts.bPressValve_Q := FALSE;
			iWorkStep := 5;
		END_IF
		IF iWorkStep <> 10 THEN fbTON_StepTimeout(IN:= FALSE); END_IF
	
	15:	// Oczekiwanie na osiąfnięcie pozycji roboczej
		IF fb2Start.bStartSig THEN
			stInOuts.bPressValve_Q := TRUE;
			IF stInOuts.bPressWorkPos THEN
				I_PimSystem.mSetNewMachineState(nPIM_MachineStates._4_OperationInProgress);
				iWorkStep := 20;
			END_IF
		ELSE
			stInOuts.bPressValve_Q := FALSE;
			mNewEvent(nEventClass:= nPIM_EventClasses.Error, nEvent:= nManometerTubeAssy_ErrorCodes.OperInteruptedBeforeWorkPos);
			// iWorkStep := 5;
		END_IF		
		fbTON_StepTimeout(IN:= TRUE, PT := T#2S);
		IF fbTON_StepTimeout.Q THEN
			mNewEvent(nEventClass:= nPIM_EventClasses.Error, nEvent:= nManometerTubeAssy_ErrorCodes.WorkPosAchieveTimeout);
		ELSIF iWorkStep <> 15 THEN fbTON_StepTimeout(IN:= FALSE); END_IF
		
	20:	// Prasa w pozycji roboczej - oczekiwanie przez zadany czas
		fbTON_StepTimeout(IN:= TRUE, PT := T#500MS);
		IF NOT stInOuts.bPressWorkPos THEN
			mNewEvent(nEventClass:= nPIM_EventClasses.Error, nEvent:= nManometerTubeAssy_ErrorCodes.WorkPosLost);
		ELSIF fbTON_StepTimeout.Q THEN
			udiOperationsOK_Qty := udiOperationsOK_Qty +1;
			I_PimSystem.mSetNewMachineState(nPIM_MachineStates._5_OperationEndedOK);
			iWorkStep := 25;
		END_IF
		IF iWorkStep <> 20 THEN	fbTON_StepTimeout(IN:= FALSE); END_IF
		
	25:	// Cofnięcie prasy
		IF I_PimSystem.mSetNewMachineState(nPIM_MachineStates._6_ReturningToBaseState) THEN
			stInOuts.bPressValve_Q := FALSE;
			iWorkStep := 30;
		END_IF

	30:	// Zakończenie operacji		 
		IF stInOuts.bPressHomePos THEN
			fbTON_StepTimeout(IN:= FALSE);
			iWorkStep := 35;
		ELSE
			fbTON_StepTimeout(IN:= TRUE, PT := T#2S);
			IF fbTON_StepTimeout.Q THEN
				mNewEvent(nEventClass:= nPIM_EventClasses.Error, nEvent:= nManometerTubeAssy_ErrorCodes.HomePosAchieveTimeout);		// Błąd powrotu do pozycji bazowej
			END_IF
		END_IF
				
	35:	// Czekanie na zwolnienie dwustartu i podniesienie uchwytu (wyciągnięcie części)
		IF NOT fb2Start.bStartSig AND NOT stInOuts.bHandleWorkPos THEN
			iWorkStep := 5;
		END_IF
		
	90:	// Zapis statusu NOK i blokowanie stanowiska
		stInOuts.bPressValve_Q := stInOuts.bPressWorkPos;
		I_PimSystem.mSetNewMachineState(nPIM_MachineStates._8_WaitForReset);
		iWorkStep := 91;
		
	91:	// Oczekiwanie na potwierdzenie
		IF I_PimSystem.mSetNewMachineState(nPIM_MachineStates._9_ResetInProgress) OR bServiceReset THEN
			bServiceReset := FALSE;
			fbTON_StepTimeout(IN:= FALSE);
			iWorkStep := 95;
		END_IF
		
	95:	// Potwierdzenie błedu
		IF NOT stInOuts.st2HandStartIO.bEmergButton_NC THEN
			mNewEvent(nEventClass:= nPIM_EventClasses.Error, nEvent:= nManometerTubeAssy_ErrorCodes.SafetySystemNotArmed);
		ELSE
			stInOuts.bPressValve_Q := FALSE;
			IF stInOuts.bPressHomePos AND stInOuts.st2HandStartIO.bEmergButton_NC AND fbTON_StepTimeout.ET > T#200MS THEN
				nError := nManometerTubeAssy_ErrorCodes.NoError;
				I_PimSystem.mSetNewMachineState(nPIM_MachineStates._0_Standby_NotReady);
				iWorkStep := 0 ;	// Powrót do kroku inicjalizacyjnego lub wskazanego w algorytmie
			END_IF
		END_IF
		fbTON_StepTimeout(IN:= TRUE, PT := T#3S);
		IF fbTON_StepTimeout.Q THEN
			mNewEvent(nEventClass:= nPIM_EventClasses.Error, nEvent:= nManometerTubeAssy_ErrorCodes.ResetTimeout);
		END_IF

	ELSE	// Krok domyślny w przypadku błędu w programie
		mNewEvent(nEventClass:= nPIM_EventClasses.Error, nEvent:= nManometerTubeAssy_ErrorCodes.ProgramConfigError);		
END_CASE
stInOuts.bPressValve_Q R= NOT stInOuts.st2HandStartIO.bEmergButton_NC;

METHOD FB_init : BOOL
VAR_INPUT
	bInitRetains : BOOL; // if TRUE, the retain variables are initialized (warm start / cold start)
	bInCopyCode : BOOL;  // if TRUE, the instance afterwards gets moved into the copy code (online change)
	I_Pim	: I_PIM;		// Interfejs do bloku PIM
END_VAR
I_PimSystem := I_Pim;
END_METHOD

(* Metoda TRUE kiedy dane wyjściowe są ok, jeśli nie FALSE (jeśli not bBusy i FALSE to błąd odczytu) *)
METHOD mGetParamsData : BOOL
VAR_INPUT
	bTestParams:	BOOL;	// Jeśli TRUE metoda okresla czy ma dostęp do parametrów, jeśli tak zwraca TRUE, jeśli nie FALSE
END_VAR
VAR_OUTPUT
	bBusy	: BOOL;										//	Maszyna odświeża dane
	pMachineParametersStruct	: POINTER TO BYTE;		// 	Wskaźnik do parametrów pracy maszyny
	uiMachineParametersSize	: UINT;						// 	Rozmiar struktury parametrów pracy maszyny [bajty]
	wActualCRC16SumInMachine	: WORD;					//	Aktualna suma CRC16 obliczona z parametrów
END_VAR
IF bTestParams THEN
	mGetParamsData := FALSE;
ELSE
	pMachineParametersStruct := 0;
	uiMachineParametersSize := 0;
	wActualCRC16SumInMachine := F_DATA_TO_CRC16_CCITT(pData := pMachineParametersStruct, cbData := uiMachineParametersSize, crc := 16#0000);
	bBusy := FALSE;
	mGetParamsData := TRUE;
END_IF
END_METHOD

METHOD INTERNAL mNewEvent : BOOL
VAR_INPUT
	nEventClass:nPIM_EventClasses;
	nEvent: nManometerTubeAssy_ErrorCodes;
END_VAR
IF nEventClass = nPIM_EventClasses.AlarmAutoConfirm OR nEventClass = nPIM_EventClasses.Message THEN		// Alarm nieblokadowy
	I_PimSystem.mSetNewMachineState(nPIM_MachineStates._0_Initialization);
	iWorkStep := 95;
ELSE
	I_PimSystem.mSetNewMachineState(nPIM_MachineStates._7_ErrorOccurr);
	I_PimSystem.mNewEvent(iEventId := nEvent, nEventType := nEventClass, tMessageTime := T#0S);
	iWorkStep := 90;
END_IF
nError := nEvent;
END_METHOD

END_FUNCTION_BLOCK

// ProdLineMachines/S02_ManometerTubeAssy/V2/fbManometerTubeAssy_V2
FUNCTION_BLOCK fbManometerTubeAssy_V2 IMPLEMENTS I_StationMachine
VAR_IN_OUT
	stInOuts: stManometerTubeAssy_V2_InOuts;
END_VAR
VAR_INPUT
	tDeltaDwuStart:TIME:= T#200MS;
END_VAR
VAR_OUTPUT
	nError:nManometerTubeAssy_V2_ErrorCodes;
END_VAR
VAR
	I_PimSystem			: I_PIM;
	fb2Start: fb2HandStartBasic;
	udiOperationsOK_Qty: UDINT;
	iWorkStep: INT;
	fbTON_StepTimeout: TON;
	fbTON_StepWaitForWorkPoss: TON;
	bServiceReset: BOOL;
	fbTON_AfterCompleteWait : TON;
	fbTON_StepColdown		: TON;
	tColdownTime			: TIME := T#150MS;
	bMinPressPosAchieved: BOOL;
END_VAR

fb2Start(stInOutsData:= stInOuts.st2HandStartIO, tDeltaDwuStart := T#250MS);

//  Błędy monitorowane stale (bezpieczeństwo)
IF NOT stInOuts.st2HandStartIO.bEmergButton_NC AND iWorkStep <> 95 AND nError <> nManometerTubeAssy_V2_ErrorCodes.SafetySystemNotArmed THEN
	stInOuts.bPressValve_Q := FALSE;
	stInOuts.bMoveValve_Q R= stInOuts.bPressHomePos;
	mNewEvent(nEvent:=nManometerTubeAssy_V2_ErrorCodes.SafetySystemNotArmed , nEventClass := nPIM_EventClasses.Error);
END_IF

CASE iWorkStep OF 
	0:	// Inicjalizacja
		I_PimSystem.mSetNewMachineState(nPIM_MachineStates._0_Initialization);
		iWorkStep := 1;
		
	1:	// Init
		I_PimSystem.mSetNewMachineState(nPIM_MachineStates._0_Standby_NotReady);
		stInOuts.bPressValve_Q := stInOuts.bMoveValve_Q := FALSE;
		iWorkStep := 5;
		
	5:	// Krok spoczynkowy - oczekiwanie na nową operację
		I_PimSystem.mSetNewMachineState(nPIM_MachineStates._2_ReadyForNewOperation);
		fbTON_AfterCompleteWait(IN:=TRUE,PT:=T#1S);
		IF fb2Start.bStartSig THEN
			IF fbTON_AfterCompleteWait.Q THEN
				IF stInOuts.bPressHomePos AND NOT stInOuts.bMoverWorkPos AND NOT stInOuts.bPressWorkPos THEN
					IF I_PimSystem.mSetNewMachineState(nPIM_MachineStates._3_NewOperationStarted) THEN 
						iWorkStep := 10;
						fbTON_StepTimeout(IN:= FALSE);
					ELSE
						mNewEvent(nEventClass:= nPIM_EventClasses.Alarm, nEvent:= nManometerTubeAssy_V2_ErrorCodes.NoWorkPermittionFromPIM);
					END_IF	
				ELSIF NOT stInOuts.bPressHomePos OR  stInOuts.bPressWorkPos THEN 
					mNewEvent(nEventClass:= nPIM_EventClasses.Alarm, nEvent:= nManometerTubeAssy_V2_ErrorCodes.PusherHomePositionError);
				ELSIF stInOuts.bMoverWorkPos THEN
					mNewEvent(nEventClass:= nPIM_EventClasses.Alarm, nEvent:= nManometerTubeAssy_V2_ErrorCodes.CartridgeHomePositionError);
				END_IF
			ELSE
				mNewEvent(nEventClass:= nPIM_EventClasses.Alarm, nEvent:= nManometerTubeAssy_V2_ErrorCodes.OperationTooEarly);			
			END_IF
		END_IF
	
	10:	// Nowa operacja rozpoczęta - ustawienie sygnałów
		IF fb2Start.bStartSig THEN
			fbTON_StepTimeout(IN:= TRUE, PT:= T#1S);
			stInOuts.bMoveValve_Q := TRUE;
			fbTON_StepColdown(IN:=stInOuts.bMoverWorkPos,PT:=tColdownTime);	//Oczekiwanie pewną ilość czasu na następny krok
			IF fbTON_StepColdown.Q THEN	// Jest ruch siłownika
				bMinPressPosAchieved := FALSE;
				fbTON_AfterCompleteWait(IN:=FALSE);
				I_PimSystem.mSetNewMachineState(nPIM_MachineStates._4_OperationInProgress);
				iWorkStep := 15;
			ELSIF fbTON_StepTimeout.Q THEN
				stInOuts.bPressValve_Q := FALSE;
				stInOuts.bMoveValve_Q R= stInOuts.bPressHomePos;
				mNewEvent(nEventClass:= nPIM_EventClasses.Alarm, nEvent:= nManometerTubeAssy_V2_ErrorCodes.CartridgeWorkPositionError);
			END_IF
		ELSE
			stInOuts.bPressValve_Q := FALSE;
			IF stInOuts.bPressHomePos THEN
				stInOuts.bMoveValve_Q := FALSE;
				iWorkStep := 5;
			END_IF
		END_IF
		IF iWorkStep <> 10 THEN fbTON_StepTimeout(IN:= FALSE);fbTON_StepColdown(IN:=FALSE); END_IF
		
	15: //Oczekiwanie na osiągnięcie przez wypychacz zadeklarowanej pozycji
		fbTON_StepTimeout(IN:= TRUE, PT := T#1S);
		stInOuts.bPressValve_Q := TRUE;
		bMinPressPosAchieved S= stInOuts.bPressWorkPos;
		fbTON_StepColdown(IN:= bMinPressPosAchieved, PT:= T#300MS);
		IF fbTON_StepColdown.Q THEN
			udiOperationsOK_Qty := udiOperationsOK_Qty +1;
			I_PimSystem.mSetNewMachineState(nPIM_MachineStates._5_OperationEndedOK);
			iWorkStep := 20;
		ELSIF fbTON_StepTimeout.Q THEN
			mNewEvent(nEventClass:= nPIM_EventClasses.Error, nEvent:= nManometerTubeAssy_V2_ErrorCodes.PusherWorkPositionError);
		END_IF
		IF iWorkStep <> 15 THEN	fbTON_StepTimeout(IN:= FALSE);fbTON_StepColdown(IN:=FALSE); END_IF
		
	20: //Oczekiwanie na wycofanie wypychacza
		fbTON_StepTimeout(IN:= TRUE, PT:= T#500MS);	
		stInOuts.bPressValve_Q := FALSE;
		IF stInOuts.bPressHomePos THEN
			iWorkStep := 25;
		ELSIF fbTON_StepTimeout.Q THEN
			mNewEvent(nEventClass:= nPIM_EventClasses.Alarm, nEvent:= nManometerTubeAssy_V2_ErrorCodes.PusherHomePositionError);
		END_IF
		IF iWorkStep <> 20 THEN	fbTON_StepTimeout(IN:= FALSE);fbTON_StepColdown(IN:=FALSE); END_IF

	25: // Sprawdzenie zezwolenia na powrót do stanu bazowego
		IF I_PimSystem.mSetNewMachineState(nPIM_MachineStates._6_ReturningToBaseState) THEN
			iWorkStep := 30;
		END_IF
		
	30: //Wywołanie wycofania siłownika z gotowym elementem
		fbTON_StepTimeout(IN:= TRUE, PT:= T#1S);	
		fbTON_StepColdown(IN:=NOT stInOuts.bMoverWorkPos, PT:= T#200MS);
		stInOuts.bMoveValve_Q R= stInOuts.bPressHomePos;
		IF fbTON_StepColdown.Q THEN
			iWorkStep := 35;
		ELSIF fbTON_StepTimeout.Q THEN
			mNewEvent(nEventClass:= nPIM_EventClasses.Alarm, nEvent:= nManometerTubeAssy_V2_ErrorCodes.CartridgeHomePositionError);	
		END_IF
		IF iWorkStep <> 30 THEN	fbTON_StepTimeout(IN:= FALSE);fbTON_StepColdown(IN:=FALSE); END_IF

	35:	// Czekanie na zwolnienie dwustartu i podniesienie uchwytu (wyciągnięcie części)
		IF NOT fb2Start.bStartSig THEN
			iWorkStep := 1;
		END_IF
//-------------------------------------------------------------------------------------------------------
	90:	// Zapis statusu NOK i blokowanie stanowiska
		I_PimSystem.mSetNewMachineState(nPIM_MachineStates._8_WaitForReset);
		iWorkStep := 91;
		
	91:	// Oczekiwanie na potwierdzenie
		IF I_PimSystem.mSetNewMachineState(nPIM_MachineStates._9_ResetInProgress) OR bServiceReset THEN
			fbTON_StepTimeout(IN:= FALSE);
			iWorkStep := 95;
		END_IF
		
	95:	// Potwierdzenie błedu
		IF NOT stInOuts.st2HandStartIO.bEmergButton_NC THEN
			mNewEvent(nEventClass:= nPIM_EventClasses.Error, nEvent:= nManometerTubeAssy_V2_ErrorCodes.SafetySystemNotArmed);
		ELSE
			stInOuts.bPressValve_Q := FALSE;
			IF stInOuts.bPressHomePos THEN
				stInOuts.bMoveValve_Q := FALSE;
			END_IF
			IF stInOuts.bPressHomePos AND stInOuts.st2HandStartIO.bEmergButton_NC AND NOT stInOuts.bMoverWorkPos AND fbTON_StepTimeout.ET > T#200MS THEN
				nError := nManometerTubeAssy_V2_ErrorCodes.NoError;
				I_PimSystem.mSetNewMachineState(nPIM_MachineStates._0_Standby_NotReady);
				iWorkStep := 1 ;	// Powrót do kroku inicjalizacyjnego lub wskazanego w algorytmie
			END_IF
		END_IF
		fbTON_StepTimeout(IN:= TRUE, PT := T#3S);
		IF fbTON_StepTimeout.Q THEN
			mNewEvent(nEventClass:= nPIM_EventClasses.Error, nEvent:= nManometerTubeAssy_V2_ErrorCodes.ResetTimeout);
		END_IF

	ELSE	// Krok domyślny w przypadku błędu w programie
		mNewEvent(nEventClass:= nPIM_EventClasses.Error, nEvent:= nManometerTubeAssy_V2_ErrorCodes.ProgramConfigError);		
END_CASE

METHOD FB_init : BOOL
VAR_INPUT
	bInitRetains : BOOL; // if TRUE, the retain variables are initialized (warm start / cold start)
	bInCopyCode : BOOL;  // if TRUE, the instance afterwards gets moved into the copy code (online change)
	I_Pim	: I_PIM;		// Interfejs do bloku PIM
END_VAR
I_PimSystem := I_Pim;
END_METHOD

(* Metoda TRUE kiedy dane wyjściowe są ok, jeśli nie FALSE (jeśli not bBusy i FALSE to błąd odczytu) *)
METHOD mGetParamsData : BOOL
VAR_INPUT
	bTestParams:	BOOL;	// Jeśli TRUE metoda okresla czy ma dostęp do parametrów, jeśli tak zwraca TRUE, jeśli nie FALSE
END_VAR
VAR_OUTPUT
	bBusy	: BOOL;										//	Maszyna odświeża dane
	pMachineParametersStruct	: POINTER TO BYTE;		// 	Wskaźnik do parametrów pracy maszyny
	uiMachineParametersSize	: UINT;						// 	Rozmiar struktury parametrów pracy maszyny [bajty]
	wActualCRC16SumInMachine	: WORD;					//	Aktualna suma CRC16 obliczona z parametrów
END_VAR
IF bTestParams THEN
	mGetParamsData := FALSE;
ELSE
	pMachineParametersStruct := 0;
	uiMachineParametersSize := 0;
	wActualCRC16SumInMachine := F_DATA_TO_CRC16_CCITT(pData := pMachineParametersStruct, cbData := uiMachineParametersSize, crc := 16#0000);
	bBusy := FALSE;
	mGetParamsData := TRUE;
END_IF
END_METHOD

METHOD INTERNAL mNewEvent : BOOL
VAR_INPUT
	nEventClass:nPIM_EventClasses;
	nEvent: nManometerTubeAssy_V2_ErrorCodes;
END_VAR
IF nEventClass = nPIM_EventClasses.AlarmAutoConfirm OR nEventClass = nPIM_EventClasses.Message THEN		// Alarm nieblokadowy
	I_PimSystem.mSetNewMachineState(nPIM_MachineStates._0_Initialization);
	iWorkStep := 95;
ELSE
	I_PimSystem.mSetNewMachineState(nPIM_MachineStates._7_ErrorOccurr);
	I_PimSystem.mNewEvent(iEventId := nEvent, nEventType := nEventClass, tMessageTime := T#0S);
	iWorkStep := 90;
END_IF
nError := nEvent;
END_METHOD

END_FUNCTION_BLOCK

// ProdLineMachines/S05_BallsWheelPress/fbBallCounterWeightPress
FUNCTION_BLOCK fbBallCounterWeightPress IMPLEMENTS I_StationMachine
VAR_IN_OUT
	stDigInOuts: stBallCounterWeightPress_InOuts;
END_VAR
VAR_INPUT
	bStartSig			: BOOL;
	stMachSettings		: stBallCounterWeightPress_Params;
END_VAR
VAR_OUTPUT
	nError:nBallCounterPressPress_ErrorCodes;
END_VAR
VAR
	I_PimSystem			: I_PIM;
	fbAlarmTab:REFERENCE TO fbAlarmSlaveTable;

	bZezwoleniePIM: BOOL;
	fbTON_Dwustart, fbTON_BladStykow:TON;
	bResetIntenal: BOOL;
	fbTON_AutoReset: TON;
	udiOperationsOK_Qty: UDINT;
	iTmp: INT;
	iWorkStep: INT;
	fbTON_StabilizerWorkPos: TON;
	fbTON_StepTimeout: TON;
	iOperationCounter: INT;
	fbTP_WibrFeederImp: TP;
	fbWheelSensorFilter: fbBinaryFilter;
	fbTON_StartDelay: TON;
	bBallsOR: BOOL;
	bBallsAND: BOOL;
	bServiceReset: BOOL;
END_VAR

// Uzupełnienie wskaźników/ danych ogólnych itp.
	
fbWheelSensorFilter(IN:= stDigInOuts.bWheelPresenceSensor, tON := T#400MS, tOFF := T#400MS);
fbTON_StartDelay(IN:= bStartSig, PT:= T#100MS);
fbTP_WibrFeederImp(IN:= FALSE, Q=> stDigInOuts.bWibrationFeeder_Q);
bBallsOR := stDigInOuts.bBallSensorInWheel[1] OR stDigInOuts.bBallSensorInWheel[2] OR stDigInOuts.bBallSensorInWheel[3];
bBallsAND := stDigInOuts.bBallSensorInWheel[1] AND stDigInOuts.bBallSensorInWheel[2] AND stDigInOuts.bBallSensorInWheel[3];

CASE iWorkStep OF 
	0:	// Inicjalizacja
		I_PimSystem.mSetNewMachineState(nPIM_MachineStates._0_Initialization);
		stDigInOuts.bPressValve_Q:= FALSE;
		iWorkStep := 1;
		
	1:	// Init
		I_PimSystem.mSetNewMachineState(nPIM_MachineStates._0_Standby_NotReady);
		iWorkStep := 5;
	
	5:	// Krok spoczynkowy - oczekiwanie na nową operację
		I_PimSystem.mSetNewMachineState(nPIM_MachineStates._2_ReadyForNewOperation);
		stDigInOuts.bPressValve_Q:= FALSE;
		IF fbTON_StartDelay.Q THEN
			IF fbWheelSensorFilter.Q AND NOT (stMachSettings.bBallsCheck AND bBallsOR) AND I_PimSystem.mSetNewMachineState(nPIM_MachineStates._3_NewOperationStarted) THEN 
				iWorkStep := 10;
				fbTON_StepTimeout(IN:= FALSE);
			ELSIF NOT fbWheelSensorFilter.Q THEN
				I_PimSystem.mNewServiceMessage(sMessage := 'Wheel not detected- operation passed',tMessageTime := T#5S);
			ELSIF stMachSettings.bBallsCheck AND bBallsOR THEN
				I_PimSystem.mNewServiceMessage(sMessage := 'Balls detected at current wheel- operation passed',tMessageTime := T#5S);	
			ELSIF NOT I_PimSystem.mSetNewMachineState(nPIM_MachineStates._3_NewOperationStarted) THEN 
				I_PimSystem.mNewServiceMessage(sMessage := 'No Work permition from PIM system',tMessageTime := T#5S);	
			END_IF
		END_IF
		
	10:	// Nowa operacja rozpoczęta - ustawienie sygnałów
		IF bStartSig THEN
			fbTON_StepTimeout(IN:= TRUE, PT := T#500MS);
			stDigInOuts.bPressValve_Q:= TRUE;
			IF NOT stDigInOuts.bPressUpPosition THEN		// Jest reakcja na sygnał startu
				iWorkStep := 15;
			ELSIF fbTON_StepTimeout.Q THEN
				mNewEvent(nEventClass:= nPIM_EventClasses.Alarm, nEvent:= nBallCounterPressPress_ErrorCodes.NoMachineReactionOnStartSig);
			END_IF
		ELSE
			stDigInOuts.bPressValve_Q:= FALSE;
			iWorkStep := 5;
		END_IF
		IF iWorkStep <> 10 THEN	fbTON_StepTimeout(IN:= FALSE); END_IF
		
	15:	// Oczekiwanie na osiągnięcie pozycji roboczej
		IF bStartSig THEN
			fbTON_StepTimeout(IN:= TRUE, PT:= T#1S);
			stDigInOuts.bPressValve_Q := TRUE;
			IF stDigInOuts.bPressDownPosition THEN	// Jest ruch siłownika
				I_PimSystem.mSetNewMachineState(nPIM_MachineStates._4_OperationInProgress);
				iWorkStep := 20;
			ELSIF fbTON_StepTimeout.Q THEN
				stDigInOuts.bPressValve_Q := FALSE;
				mNewEvent(nEventClass:= nPIM_EventClasses.Alarm, nEvent:= nBallCounterPressPress_ErrorCodes.WorkPosAchieveTimeout);
			END_IF
		ELSE
			stDigInOuts.bPressValve_Q := FALSE;
			iWorkStep := 5;
		END_IF
		IF iWorkStep <> 15 THEN fbTON_StepTimeout(IN:= FALSE); END_IF
	
	20:	// Sprawdzenie wprasowania kulek
		fbTON_StepTimeout(IN:= TRUE, PT := T#500MS);
		IF NOT stDigInOuts.bPressDownPosition THEN
			mNewEvent(nEventClass:= nPIM_EventClasses.Alarm, nEvent:= nBallCounterPressPress_ErrorCodes.WorkPosLost);
		ELSIF fbTON_StepTimeout.Q THEN
			IF NOT stMachSettings.bBallsCheck OR bBallsAND THEN	// Wszystkie przeciwwagi są w kole
				iOperationCounter:= iOperationCounter +1;
				I_PimSystem.mSetNewMachineState(nPIM_MachineStates._5_OperationEndedOK);
				iWorkStep := 25;
			ELSE
				mNewEvent(nEventClass:= nPIM_EventClasses.Alarm, nEvent:= nBallCounterPressPress_ErrorCodes.BallsNotPresentAfterPushing);
			END_IF
		END_IF
		IF iWorkStep <> 20 THEN fbTON_StepTimeout(IN:= FALSE); END_IF
				
	25:	// Cofnięcie prasy
		IF I_PimSystem.mSetNewMachineState(nPIM_MachineStates._6_ReturningToBaseState) THEN
			stDigInOuts.bPressValve_Q := FALSE;
			iWorkStep := 30;
		END_IF

	30:	// Zakończenie operacji		 
		IF stDigInOuts.bPressUpPosition THEN
			fbTON_StepTimeout(IN:= FALSE);
			iWorkStep := 34;
		ELSE
			stDigInOuts.bPressValve_Q := FALSE;
			fbTON_StepTimeout(IN:= TRUE, PT := T#2S);
			IF fbTON_StepTimeout.Q THEN
				mNewEvent(nEventClass:= nPIM_EventClasses.Error, nEvent:= nBallCounterPressPress_ErrorCodes.HomePosAchieveTimeout);		// Błąd powrotu do pozycji bazowej
			END_IF
		END_IF
		
	34: // Start podajnika wibracyjnego
		IF stMachSettings.iEnFeederEveryNCycles > 0 AND iOperationCounter > stMachSettings.iEnFeederEveryNCycles THEN
			fbTP_WibrFeederImp(IN:= TRUE, PT:= REAL_TO_TIME(stMachSettings.rFeederOnTime_S)*1000);
			iOperationCounter := 0;
		END_IF
		iWorkStep := 35;
				
	35:	// Czekanie na zwolnienie dwustartu i podniesienie uchwytu (wyciągnięcie części)
		IF NOT bStartSig AND NOT fbWheelSensorFilter.Q THEN
			iWorkStep := 5;
			I_PimSystem.mNewServiceMessage(sMessage := '',tMessageTime := T#0S);
		ELSE
			I_PimSystem.mNewServiceMessage(sMessage := 'Waiting for start signal and wheel presence signal reset',tMessageTime := T#5S);
		END_IF
		
	90:	// Zapis statusu NOK i blokowanie stanowiska
		stDigInOuts.bPressValve_Q := stDigInOuts.bPressDownPosition;
		I_PimSystem.mSetNewMachineState(nPIM_MachineStates._8_WaitForReset);
		iWorkStep := 91;
		
	91:	// Oczekiwanie na potwierdzenie
		IF I_PimSystem.mSetNewMachineState(nPIM_MachineStates._9_ResetInProgress) OR bServiceReset THEN
			fbTON_StepTimeout(IN:= FALSE);
			iWorkStep := 95;
		END_IF
		
	95:	// Potwierdzenie błedu
		stDigInOuts.bPressValve_Q := FALSE;
		IF stDigInOuts.bPressUpPosition AND fbTON_StepTimeout.ET > T#200MS THEN
			nError := nBallCounterPressPress_ErrorCodes.NoError;
			I_PimSystem.mSetNewMachineState(nPIM_MachineStates._0_Standby_NotReady);
			iWorkStep := 0 ;	// Powrót do kroku inicjalizacyjnego lub wskazanego w algorytmie
		END_IF
		fbTON_StepTimeout(IN:= TRUE, PT := T#3S);
		IF fbTON_StepTimeout.Q THEN
			mNewEvent(nEventClass:= nPIM_EventClasses.Error, nEvent:= nBallCounterPressPress_ErrorCodes.ResetTimeout);
		END_IF

	ELSE	// Krok domyślny w przypadku błędu w programie
		mNewEvent(nEventClass:= nPIM_EventClasses.Error, nEvent:= nBallCounterPressPress_ErrorCodes.ProgramConfigError);		
END_CASE

METHOD FB_init : BOOL
VAR_INPUT
	bInitRetains : BOOL; // if TRUE, the retain variables are initialized (warm start / cold start)
	bInCopyCode : BOOL;  // if TRUE, the instance afterwards gets moved into the copy code (online change)
	I_Pim	: I_PIM;		// Interfejs do bloku PIM
END_VAR
I_PimSystem := I_Pim;
END_METHOD

(* Metoda TRUE kiedy dane wyjściowe są ok, jeśli nie FALSE (jeśli not bBusy i FALSE to błąd odczytu) *)
METHOD mGetParamsData : BOOL
VAR_INPUT
	bTestParams:	BOOL;	// Jeśli TRUE metoda okresla czy ma dostęp do parametrów, jeśli tak zwraca TRUE, jeśli nie FALSE
END_VAR
VAR_OUTPUT
	bBusy	: BOOL;										//	Maszyna odświeża dane
	pMachineParametersStruct	: POINTER TO BYTE;		// 	Wskaźnik do parametrów pracy maszyny
	uiMachineParametersSize	: UINT;						// 	Rozmiar struktury parametrów pracy maszyny [bajty]
	wActualCRC16SumInMachine	: WORD;					//	Aktualna suma CRC16 obliczona z parametrów
END_VAR
IF bTestParams THEN
	mGetParamsData := FALSE;
ELSE
	pMachineParametersStruct := 0;
	uiMachineParametersSize := 0;
	wActualCRC16SumInMachine := F_DATA_TO_CRC16_CCITT(pData := pMachineParametersStruct, cbData := uiMachineParametersSize, crc := 16#0000);
	bBusy := FALSE;
	mGetParamsData := TRUE;
END_IF
END_METHOD

METHOD INTERNAL mNewEvent : BOOL
VAR_INPUT
	nEventClass:nPIM_EventClasses;
	nEvent: nBallCounterPressPress_ErrorCodes;
END_VAR
IF nEventClass = nPIM_EventClasses.AlarmAutoConfirm OR nEventClass = nPIM_EventClasses.Message THEN		// Alarm nieblokadowy
	I_PimSystem.mSetNewMachineState(nPIM_MachineStates._0_Initialization);
	iWorkStep := 95;
ELSE
	I_PimSystem.mSetNewMachineState(nPIM_MachineStates._7_ErrorOccurr);
	I_PimSystem.mNewEvent(iEventId := nEvent, nEventType := nEventClass, tMessageTime := T#0S);
	iWorkStep := 90;
END_IF
nError := nEvent;
END_METHOD

END_FUNCTION_BLOCK

// ProdLineMachines/S11_ResWelderTecna/fbTecnaResWelder
FUNCTION_BLOCK fbTecnaResWelder IMPLEMENTS I_StationMachine
VAR_IN_OUT
	stInOuts: stTecnaResWelder_InOuts;
END_VAR
VAR_OUTPUT
	nError 				: nTecnaResWelder_ErrorCodes;
END_VAR
VAR
	I_PimSystem			: I_PIM;
	iWorkStep: INT;
	bServiceReset: BOOL;
	bRightSideWelded: BOOL;
	bLeftSideWelded: BOOL;
	iSyncError: INT;
	iLeftSensorWorkCheck, iRightSensorWorkCheck: INT;
	fbLeftMotorSensor, fbRightMotorSensor, fbEndCycle: fbBinaryFilter;
	bReworkON: BOOL;				//Zmienna dla obsługi trybu REwork przy zastosowaniu zmiennych parametrów;
	iReturnToWorkStep: INT;
	iNokReporteds: INT;
	fbFTRIG_UserLogin: F_TRIG;
END_VAR
VAR PERSISTENT
	stWorkParams	: stTecnaResWelder_TestParams;
END_VAR

// Signals preparation
stInOuts.bWorkPermission_Q := I_PimSystem.prWorkPermission AND iWorkStep < 90;
fbLeftMotorSensor(IN:= stInOuts.bLeftMotorSensor, tON := T#250MS, tOFF := T#1S);
fbRightMotorSensor(IN:= stInOuts.bRightMotorSensor, tON := T#250MS, tOFF := T#1S);
fbEndCycle(IN:= stInOuts.bEndCycle, tON := T#0MS, tOFF := T#200MS, bReset := FALSE);
fbFTRIG_UserLogin(CLK:= I_PimSystem.prUserLogged);

IF I_PimSystem.prNokReportedSource = nPIM_ReportedNokSource.FromMach THEN
	IF stWorkParams.bResetWhenNokReported THEN
		iReturnToWorkStep := 1;
		iWorkStep := 1;
	ELSE
		iNokReporteds:= iNokReporteds + 1; 
	END_IF
ELSIF fbFTRIG_UserLogin.Q THEN 
		iReturnToWorkStep := 1;
		iWorkStep := 1;	
END_IF

IF fbLeftMotorSensor.FTrig THEN
	iLeftSensorWorkCheck := 0;
END_IF
IF fbRightMotorSensor.FTrig THEN
	iRightSensorWorkCheck := 0;
END_IF
 

// Rework mode (diferent program for left and right weld) ------------------------------------------------------
stInOuts.bProgramChange := stWorkParams.bReworkMode_EN AND stInOuts.bLeftMotorSensor;


//------------------------------------------------------
CASE iWorkStep OF 
	0:	// Inicjalizacja
		I_PimSystem.mSetNewMachineState(nPIM_MachineStates._0_Initialization);
		iWorkStep := 1;
		
	1:	// Init
		I_PimSystem.mSetNewMachineState(nPIM_MachineStates._0_Standby_NotReady);
		bRightSideWelded := bLeftSideWelded := FALSE;
		iWorkStep := 5;
	
	5:	// Krok spoczynkowy - oczekiwanie na nową operację
		I_PimSystem.mSetNewMachineState(nPIM_MachineStates._2_ReadyForNewOperation);
		IF fbEndCycle.RTrig THEN	// Nowy zgrzew 
			IF I_PimSystem.mSetNewMachineState(nPIM_MachineStates._3_NewOperationStarted) THEN 
				IF stWorkParams.bCheckWeldsOrder THEN	
					IF iLeftSensorWorkCheck > 3 OR iRightSensorWorkCheck > 3 OR (fbLeftMotorSensor.Q AND fbRightMotorSensor.Q) THEN	// Sensor errors
						mNewEvent(nEventClass := nPIM_EventClasses.Error, nEvent := nTecnaResWelder_ErrorCodes.SensorWorkError);
					ELSIF fbLeftMotorSensor.Q AND NOT fbRightMotorSensor.Q THEN	// Sytuacja ok
						iLeftSensorWorkCheck := iLeftSensorWorkCheck + 1;
						bLeftSideWelded := TRUE;
						iWorkStep := 10;
					ELSIF NOT fbLeftMotorSensor.Q AND fbRightMotorSensor.Q THEN	// Niewłaściwa strona
						mNewEvent(nEventClass := nPIM_EventClasses.Error, nEvent := nTecnaResWelder_ErrorCodes.InvalidWeldOrder_FirstLeft);
					ELSE
						mNewEvent(nEventClass := nPIM_EventClasses.Alarm, nEvent := nTecnaResWelder_ErrorCodes.NoPartDetected);	
					END_IF
				ELSE
					IF fbLeftMotorSensor.Q THEN
						bLeftSideWelded := TRUE;	
						iLeftSensorWorkCheck := iLeftSensorWorkCheck + 1;
					END_IF
					IF fbRightMotorSensor.Q THEN
						bRightSideWelded := TRUE;	
						iRightSensorWorkCheck := iRightSensorWorkCheck + 1;
					END_IF
					iWorkStep := 10;	
				END_IF
			ELSE
				I_PimSystem.mNewServiceMessage(sMessage := 'No Work permition from PIM system- part missed',tMessageTime := T#5S);	
			END_IF
		END_IF
		
	10:	// Nowa operacja rozpoczęta - ustawienie sygnałów
		I_PimSystem.mSetNewMachineState(nPIM_MachineStates._4_OperationInProgress);
		iWorkStep := 15;
	
	15:	// Oczekiwanie na osiągnięcie pozycji roboczej
		IF fbEndCycle.RTrig THEN
			IF stWorkParams.bCheckWeldsOrder THEN	
				IF fbLeftMotorSensor.Q AND fbRightMotorSensor.Q THEN	// Sensor errors
					mNewEvent(nEventClass := nPIM_EventClasses.Error, nEvent := nTecnaResWelder_ErrorCodes.SensorWorkError);
				ELSIF NOT fbLeftMotorSensor.Q AND fbRightMotorSensor.Q THEN	// Sytuacja ok
					iRightSensorWorkCheck := iRightSensorWorkCheck + 1;
					bRightSideWelded := TRUE;
					iWorkStep := 20;
				ELSIF fbLeftMotorSensor.Q AND NOT fbRightMotorSensor.Q THEN	// Niewłaściwa strona
					mNewEvent(nEventClass := nPIM_EventClasses.Error, nEvent := nTecnaResWelder_ErrorCodes.InvalidWeldOrder_FirstLeft);
				ELSE
					iReturnToWorkStep := iWorkStep;
					mNewEvent(nEventClass := nPIM_EventClasses.Error, nEvent := nTecnaResWelder_ErrorCodes.NoPartDetected);	
				END_IF
			ELSE
				IF fbLeftMotorSensor.Q THEN
					bLeftSideWelded := TRUE;	
					iLeftSensorWorkCheck := iLeftSensorWorkCheck + 1;
				END_IF
				IF fbRightMotorSensor.Q THEN
					bRightSideWelded := TRUE;	
					iRightSensorWorkCheck := iRightSensorWorkCheck + 1;
				END_IF
				iWorkStep := 20;	
			END_IF
		END_IF
		
	20:	// Sprawdzenie czy zgrzano silnik z dwóch stron	
		IF NOT bRightSideWelded OR NOT bLeftSideWelded THEN
			iSyncError := iSyncError +1; 
		END_IF			
		I_PimSystem.mSetNewMachineState(nPIM_MachineStates._5_OperationEndedOK);
		iWorkStep := 25;
		
	25:	// Cofnięcie prasy
		IF I_PimSystem.mSetNewMachineState(nPIM_MachineStates._6_ReturningToBaseState) THEN
			iWorkStep := 30;
		END_IF

	30:	// Zakończenie operacji		 
		IF NOT fbLeftMotorSensor.Q AND NOT fbRightMotorSensor.Q THEN
			iWorkStep := 1;
		ELSIF fbEndCycle.RTrig AND stWorkParams.bCheckWeldsOrder THEN
			mNewEvent(nEventClass := nPIM_EventClasses.Alarm, nEvent := nTecnaResWelder_ErrorCodes.SensorWorkError);
		END_IF
				
		
	90:	// Zapis statusu NOK i blokowanie stanowiska
		I_PimSystem.mSetNewMachineState(nPIM_MachineStates._8_WaitForReset);
		iWorkStep := 91;
		
	91:	// Oczekiwanie na potwierdzenie
		IF I_PimSystem.mSetNewMachineState(nPIM_MachineStates._9_ResetInProgress) OR bServiceReset THEN
			bServiceReset := FALSE;
			iWorkStep := 95;
		END_IF
		
	95:	// Potwierdzenie błedu
		I_PimSystem.mSetNewMachineState(nPIM_MachineStates._0_Standby_NotReady);
		nError := nTecnaResWelder_ErrorCodes.NoError;
		iWorkStep := iReturnToWorkStep;	// Powrót do kroku inicjalizacyjnego lub wskazanego w algorytmie
		iReturnToWorkStep := 1;
END_CASE

METHOD FB_init : BOOL
VAR_INPUT
	bInitRetains : BOOL; // if TRUE, the retain variables are initialized (warm start / cold start)
	bInCopyCode : BOOL;  // if TRUE, the instance afterwards gets moved into the copy code (online change)
	I_Pim	: I_PIM;		// Interfejs do bloku PIM
END_VAR
I_PimSystem := I_Pim;
END_METHOD

(* Metoda TRUE kiedy dane wyjściowe są ok, jeśli nie FALSE (jeśli not bBusy i FALSE to błąd odczytu) *)
METHOD mGetParamsData : BOOL
VAR_INPUT
	bTestParams:	BOOL;	// Jeśli TRUE metoda okresla czy ma dostęp do parametrów, jeśli tak zwraca TRUE, jeśli nie FALSE
END_VAR
VAR_OUTPUT
	bBusy	: BOOL;										//	Maszyna odświeża dane
	pMachineParametersStruct	: POINTER TO BYTE;		// 	Wskaźnik do parametrów pracy maszyny
	uiMachineParametersSize	: UINT;						// 	Rozmiar struktury parametrów pracy maszyny [bajty]
	wActualCRC16SumInMachine	: WORD;					//	Aktualna suma CRC16 obliczona z parametrów
END_VAR
IF bTestParams THEN
	mGetParamsData := FALSE;
ELSE
	pMachineParametersStruct := 0;
	uiMachineParametersSize := 0;
	wActualCRC16SumInMachine := F_DATA_TO_CRC16_CCITT(pData := pMachineParametersStruct, cbData := uiMachineParametersSize, crc := 16#0000);
	bBusy := FALSE;
	mGetParamsData := TRUE;
END_IF
END_METHOD

METHOD INTERNAL mNewEvent : BOOL
VAR_INPUT
	nEventClass:nPIM_EventClasses;
	nEvent: nTecnaResWelder_ErrorCodes;
END_VAR
IF nEventClass = nPIM_EventClasses.AlarmAutoConfirm OR nEventClass = nPIM_EventClasses.Message THEN		// Alarm nieblokadowy
	I_PimSystem.mSetNewMachineState(nPIM_MachineStates._0_Initialization);
	iWorkStep := 95;
ELSE
	I_PimSystem.mSetNewMachineState(nPIM_MachineStates._7_ErrorOccurr);
	I_PimSystem.mNewEvent(iEventId := nEvent, nEventType := nEventClass, tMessageTime := T#0S);
	iWorkStep := 90;
END_IF
nError := nEvent;
END_METHOD

END_FUNCTION_BLOCK

// ProdLineMachines/S12_Hios/fbHIOS_ScrewDriver
{attribute 'reflection'}
FUNCTION_BLOCK fbHIOS_ScrewDriver IMPLEMENTS I_StationMachine
VAR_IN_OUT
	stDigInOuts: stHIOS_InOuts;
END_VAR
VAR_INPUT
	stTestParam: stHIOS_TestParameters;
END_VAR
VAR_OUTPUT
	bWkretakZablokowany		:BOOL;		// Praca wkrętaka zablokowana
	bWkretakWlaczony		:BOOL;		// Wkrętak uruchomiony
	bScrewPass				:BOOL;		// Śruba wkręcona OK
	bScrewFail				:BOOL;		// Śruba wkręcona NOK
	bTorqueUp				:BOOL;		// Ustawiony moment osiągnięty
	nError					:nHIOS_ErrorList;
END_VAR
VAR
	I_PimSystem			: I_PIM;
	sVersionType: STRING(36);
	stScrewDriverParamsAct:stHIOS_ScrewDriverParams;
	fbMotorSensorFilter:fbBinaryFilter;
	fbTON_StepTimeout: TON;
	bScrewsQuantityCHanged: BOOL;
	bOczekiwanieNaOdpowiedz: BOOL;
	stFastenPIM_Data:stHIOS_FastenExtData;
	fbSendString:SendString;	
	fbRecvString:ReceiveString;	
	sSendStringfb		:STRING;
	fbTON_Timer_Comm	:TON;
	bQBladKomunikacji	:BOOL;			// Flaga oznacza, że ostatnia odpowiedź była będna lub jej nie było 
	bOdczytOK 			:BOOL;			// Odczyt ok.
	bSendString: BOOL;
	sSendingString : STRING;
	sRcvString: STRING;
	iComSendError: Tc2_SerialCom.ComError_t;
	iTypZapytanie: INT;
	sStringToRead: STRING(30);
	iActPulses: INT;
	iFailPulses: INT;
	iPassPulses: INT;
	asComunicationHistoryOut: ARRAY [1..10] OF STRING(10);
	asComunicationHistoryIn: ARRAY [1..10] OF STRING(10);
	bMaintenanceRequest: BOOL;
	sErrorString: STRING(255);
	diStartsUpCtr: DINT;
	
	fbFTRIG_UpdateMachineParams: F_TRIG;
	bReadMachineParams: BOOL;
	bWaitForAllParams: BOOL;
	iParamsCtr: INT;
	fbTON_ParamsRead: TON;
	iWorkStep: INT;	

	fbRTRIG_NewSerialCmd: R_TRIG;
	udiNbOfSavedOkStatuses,	udiNbOfSavedNokStatuses, udiNbOfSavedOkStatusesMEM, udiNbOfSavedNokStatusesMEM: UDINT;	// Liczniki zapusanych statusów PIM
	bUserLogged: BOOL;
	fbRtrig_UserLogged: R_TRIG;
	bWorkPermitt: BOOL;
	bServiceReset: BOOL;
	bSqlExtDataSave: BOOL;					// Bit ustawiany po operacji oznacza, że trzeba dane rozszerzone, resetowany po udanym lub błędnym zapisie
	astExtData: ARRAY [1..2] OF stPIM_ExtDataRow;
	bSqlExtDataSavedOK: BOOL;
	
END_VAR

// Filtrowanie sygnału obeności kompresora w kowadle - sygnał ustawiany gdy jest sygnał z czujnika jest przez tInputFlterTime, resetowany podobnie
fbMotorSensorFilter(IN:= stDigInOuts.bMotorSensor, tON:= T#300MS, tOFF := T#300MS);

I_PimSystem.mGetStationData(bUserLogged => bUserLogged, bWorkPermittion => bWorkPermitt);
fbRtrig_UserLogged(CLK:= bUserLogged);

CASE iWorkStep OF 
	0:	// Inicjalizacja
		I_PimSystem.mSetNewMachineState(nPIM_MachineStates._0_Initialization);
		iWorkStep := 1;
	
	1: // Przygotowanie do uruchomienia
		I_PimSystem.mSetNewMachineState(nPIM_MachineStates._0_Standby_NotReady);
		fbTON_StepTimeout(IN:= FALSE);
		iWorkStep := 5;
	
	5:	// Krok spoczynkowy - oczekiwanie na nową operację
		I_PimSystem.mSetNewMachineState(nPIM_MachineStates._2_ReadyForNewOperation);
		IF fbMotorSensorFilter.RTrig AND bWorkPermitt THEN
			IF I_PimSystem.mSetNewMachineState(nPIM_MachineStates._3_NewOperationStarted) THEN 
				IF bWkretakZablokowany AND NOT bOczekiwanieNaOdpowiedz AND NOT bOdczytOK THEN
					iTypZapytanie := 7;	// Odblokowanie wkrętaka gdy jest zezwolnie, a wkrętak zablokowany
				END_IF
				iWorkStep := 10;
				fbTON_StepTimeout(IN:= FALSE);
				stDigInOuts.bMotorLockValve_Q := TRUE;
				iTypZapytanie := 5;		// Reset licznika we wkrętaku
				MEMSET(destAddr := ADR(stFastenPIM_Data), n := SIZEOF(stFastenPIM_Data), fillByte := 0);
			END_IF
		ELSIF NOT bWorkPermitt AND NOT bWkretakZablokowany AND NOT bOczekiwanieNaOdpowiedz AND NOT bOdczytOK THEN
			iTypZapytanie := 6; // Jeśli wkrętak uruchomiony i brak zezwolenia na prace zablokuj
		ELSIF bWorkPermitt AND bWkretakZablokowany AND NOT bOczekiwanieNaOdpowiedz AND NOT bOdczytOK THEN
			iTypZapytanie := 7; // Odblokuj wkrętak
		END_IF
		
